   1:  PR[91,1] = PR[90,1] + 32.337;
   1:  PR[91,2] = PR[90,2] + -10.295;
   1:  PR[91,3] = PR[90,3] + 13.551;
   1:L PR[91] R[100]mm/sec CNT100;
   1:  PR[91,1] = PR[90,1] + 32.852;
   1:  PR[91,2] = PR[90,2] + -9.634;
   1:  PR[91,3] = PR[90,3] + 13.557;
   1:L PR[91] R[100]mm/sec CNT100;
   1:  PR[91,1] = PR[90,1] + 33.339;
   1:  PR[91,2] = PR[90,2] + -8.939;
   1:  PR[91,3] = PR[90,3] + 13.562;
   1:L PR[91] R[100]mm/sec CNT100;
   1:  PR[91,1] = PR[90,1] + 33.788;
   1:  PR[91,2] = PR[90,2] + -8.227;
   1:  PR[91,3] = PR[90,3] + 13.568;
   1:L PR[91] R[100]mm/sec CNT100;
   1:  PR[91,1] = PR[90,1] + 34.186;
   1:  PR[91,2] = PR[90,2] + -7.524;
   1:  PR[91,3] = PR[90,3] + 13.574;
   1:L PR[91] R[100]mm/sec CNT100;
   1:  PR[91,1] = PR[90,1] + 34.560;
   1:  PR[91,2] = PR[90,2] + -6.785;
   1:  PR[91,3] = PR[90,3] + 13.579;
   1:L PR[91] R[100]mm/sec CNT100;
   1:  PR[91,1] = PR[90,1] + 34.896;
   1:  PR[91,2] = PR[90,2] + -6.031;
   1:  PR[91,3] = PR[90,3] + 13.584;
   1:L PR[91] R[100]mm/sec CNT100;
   1:  PR[91,1] = PR[90,1] + 35.196;
   1:  PR[91,2] = PR[90,2] + -5.265;
   1:  PR[91,3] = PR[90,3] + 13.590;
   1:L PR[91] R[100]mm/sec CNT100;
   1:  PR[91,1] = PR[90,1] + 35.456;
   1:  PR[91,2] = PR[90,2] + -4.487;
   1:  PR[91,3] = PR[90,3] + 13.595;
   1:L PR[91] R[100]mm/sec CNT100;
   1:  PR[91,1] = PR[90,1] + 35.678;
   1:  PR[91,2] = PR[90,2] + -3.699;
   1:  PR[91,3] = PR[90,3] + 13.600;
   1:L PR[91] R[100]mm/sec CNT100;
   1:  PR[91,1] = PR[90,1] + 35.861;
   1:  PR[91,2] = PR[90,2] + -2.900;
   1:  PR[91,3] = PR[90,3] + 13.606;
   1:L PR[91] R[100]mm/sec CNT100;
   1:  PR[91,1] = PR[90,1] + 36.003;
   1:  PR[91,2] = PR[90,2] + -2.088;
   1:  PR[91,3] = PR[90,3] + 13.611;
   1:L PR[91] R[100]mm/sec CNT100;
   1:  PR[91,1] = PR[90,1] + 36.105;
   1:  PR[91,2] = PR[90,2] + -1.263;
   1:  PR[91,3] = PR[90,3] + 13.617;
   1:L PR[91] R[100]mm/sec CNT100;
   1:  PR[91,1] = PR[90,1] + 36.167;
   1:  PR[91,2] = PR[90,2] + -0.424;
   1:  PR[91,3] = PR[90,3] + 13.622;
   1:L PR[91] R[100]mm/sec CNT100;
   1:  PR[91,1] = PR[90,1] + 36.190;
   1:  PR[91,2] = PR[90,2] + 0.428;
   1:  PR[91,3] = PR[90,3] + 13.628;
   1:L PR[91] R[100]mm/sec CNT100;
   1:  PR[91,1] = PR[90,1] + 36.167;
   1:  PR[91,2] = PR[90,2] + 1.279;
   1:  PR[91,3] = PR[90,3] + 13.633;
   1:L PR[91] R[100]mm/sec CNT100;
   1:  PR[91,1] = PR[90,1] + 36.105;
   1:  PR[91,2] = PR[90,2] + 2.119;
   1:  PR[91,3] = PR[90,3] + 13.639;
   1:L PR[91] R[100]mm/sec CNT100;
   1:  PR[91,1] = PR[90,1] + 36.003;
   1:  PR[91,2] = PR[90,2] + 2.943;
   1:  PR[91,3] = PR[90,3] + 13.644;
   1:L PR[91] R[100]mm/sec CNT100;
   1:  PR[91,1] = PR[90,1] + 35.861;
   1:  PR[91,2] = PR[90,2] + 3.755;
   1:  PR[91,3] = PR[90,3] + 13.650;
   1:L PR[91] R[100]mm/sec CNT100;
   1:  PR[91,1] = PR[90,1] + 35.678;
   1:  PR[91,2] = PR[90,2] + 4.554;
   1:  PR[91,3] = PR[90,3] + 13.655;
   1:L PR[91] R[100]mm/sec CNT100;
   1:  PR[91,1] = PR[90,1] + 35.456;
   1:  PR[91,2] = PR[90,2] + 5.343;
   1:  PR[91,3] = PR[90,3] + 13.660;
   1:L PR[91] R[100]mm/sec CNT100;
   1:  PR[91,1] = PR[90,1] + 35.196;
   1:  PR[91,2] = PR[90,2] + 6.120;
   1:  PR[91,3] = PR[90,3] + 13.666;
   1:L PR[91] R[100]mm/sec CNT100;
   1:  PR[91,1] = PR[90,1] + 34.896;
   1:  PR[91,2] = PR[90,2] + 6.886;
   1:  PR[91,3] = PR[90,3] + 13.671;
   1:L PR[91] R[100]mm/sec CNT100;
   1:  PR[91,1] = PR[90,1] + 34.559;
   1:  PR[91,2] = PR[90,2] + 7.640;
   1:  PR[91,3] = PR[90,3] + 13.677;
   1:L PR[91] R[100]mm/sec CNT100;
   1:  PR[91,1] = PR[90,1] + 34.186;
   1:  PR[91,2] = PR[90,2] + 8.379;
   1:  PR[91,3] = PR[90,3] + 13.682;
   1:L PR[91] R[100]mm/sec CNT100;
   1:  PR[91,1] = PR[90,1] + 33.778;
   1:  PR[91,2] = PR[90,2] + 9.100;
   1:  PR[91,3] = PR[90,3] + 13.687;
   1:L PR[91] R[100]mm/sec CNT100;
   1:  PR[91,1] = PR[90,1] + 33.333;
   1:  PR[91,2] = PR[90,2] + 9.803;
   1:  PR[91,3] = PR[90,3] + 13.693;
   1:L PR[91] R[100]mm/sec CNT100;
   1:  PR[91,1] = PR[90,1] + 32.852;
   1:  PR[91,2] = PR[90,2] + 10.489;
   1:  PR[91,3] = PR[90,3] + 13.698;
   1:L PR[91] R[100]mm/sec CNT100;
   1:  PR[91,1] = PR[90,1] + 32.337;
   1:  PR[91,2] = PR[90,2] + 11.150;
   1:  PR[91,3] = PR[90,3] + 13.704;
   1:L PR[91] R[100]mm/sec CNT100;
   1:  PR[91,1] = PR[90,1] + 31.789;
   1:  PR[91,2] = PR[90,2] + 11.786;
   1:  PR[91,3] = PR[90,3] + 13.709;
   1:L PR[91] R[100]mm/sec CNT100;
   1:  PR[91,1] = PR[90,1] + 31.210;
   1:  PR[91,2] = PR[90,2] + 12.395;
   1:  PR[91,3] = PR[90,3] + 13.715;
   1:L PR[91] R[100]mm/sec CNT100;
   1:  PR[91,1] = PR[90,1] + 30.601;
   1:  PR[91,2] = PR[90,2] + 12.975;
   1:  PR[91,3] = PR[90,3] + 13.720;
   1:L PR[91] R[100]mm/sec CNT100;
   1:  PR[91,1] = PR[90,1] + 29.964;
   1:  PR[91,2] = PR[90,2] + 13.525;
   1:  PR[91,3] = PR[90,3] + 13.726;
   1:L PR[91] R[100]mm/sec CNT100;
   1:  PR[91,1] = PR[90,1] + 29.298;
   1:  PR[91,2] = PR[90,2] + 14.044;
   1:  PR[91,3] = PR[90,3] + 13.731;
   1:L PR[91] R[100]mm/sec CNT100;
   1:  PR[91,1] = PR[90,1] + 28.607;
   1:  PR[91,2] = PR[90,2] + 14.531;
   1:  PR[91,3] = PR[90,3] + 13.737;
   1:L PR[91] R[100]mm/sec CNT100;
   1:  PR[91,1] = PR[90,1] + 27.892;
   1:  PR[91,2] = PR[90,2] + 14.985;
   1:  PR[91,3] = PR[90,3] + 13.742;
   1:L PR[91] R[100]mm/sec CNT100;
   1:  PR[91,1] = PR[90,1] + 27.152;
   1:  PR[91,2] = PR[90,2] + 15.405;
   1:  PR[91,3] = PR[90,3] + 13.748;
   1:L PR[91] R[100]mm/sec CNT100;
   1:  PR[91,1] = PR[90,1] + 26.864;
   1:  PR[91,2] = PR[90,2] + 15.553;
   1:  PR[91,3] = PR[90,3] + 13.753;
   1:L PR[91] R[100]mm/sec CNT100;
   1:  PR[91,1] = PR[90,1] + 26.394;
   1:  PR[91,2] = PR[90,2] + 15.789;
   1:  PR[91,3] = PR[90,3] + 13.756;
   1:L PR[91] R[100]mm/sec CNT100;
   1:  PR[91,1] = PR[90,1] + 25.614;
   1:  PR[91,2] = PR[90,2] + 16.137;
   1:  PR[91,3] = PR[90,3] + 13.759;
   1:L PR[91] R[100]mm/sec CNT100;
   1:  PR[91,1] = PR[90,1] + 24.816;
   1:  PR[91,2] = PR[90,2] + 16.448;
   1:  PR[91,3] = PR[90,3] + 13.765;
   1:L PR[91] R[100]mm/sec CNT100;
   1:  PR[91,1] = PR[90,1] + 24.003;
   1:  PR[91,2] = PR[90,2] + 16.721;
   1:  PR[91,3] = PR[90,3] + 13.770;
   1:L PR[91] R[100]mm/sec CNT100;
   1:  PR[91,1] = PR[90,1] + 23.176;
   1:  PR[91,2] = PR[90,2] + 16.954;
   1:  PR[91,3] = PR[90,3] + 13.776;
   1:L PR[91] R[100]mm/sec CNT100;
   1:  PR[91,1] = PR[90,1] + 22.334;
   1:  PR[91,2] = PR[90,2] + 17.149;
   1:  PR[91,3] = PR[90,3] + 13.781;
   1:L PR[91] R[100]mm/sec CNT100;
   1:  PR[91,1] = PR[90,1] + 21.481;
   1:  PR[91,2] = PR[90,2] + 17.302;
   1:  PR[91,3] = PR[90,3] + 13.787;
   1:L PR[91] R[100]mm/sec CNT100;
   1:  PR[91,1] = PR[90,1] + 20.619;
   1:  PR[91,2] = PR[90,2] + 17.414;
   1:  PR[91,3] = PR[90,3] + 13.793;
   1:L PR[91] R[100]mm/sec CNT100;
   1:  PR[91,1] = PR[90,1] + 20.067;
   1:  PR[91,2] = PR[90,2] + 17.460;
   1:  PR[91,3] = PR[90,3] + 13.799;
   1:L PR[91] R[100]mm/sec CNT100;
   1:  PR[91,1] = PR[90,1] + 19.753;
   1:  PR[91,2] = PR[90,2] + 17.485;
   1:  PR[91,3] = PR[90,3] + 13.802;
   1:L PR[91] R[100]mm/sec CNT100;
   1:  PR[91,1] = PR[90,1] + 18.879;
   1:  PR[91,2] = PR[90,2] + 17.513;
   1:  PR[91,3] = PR[90,3] + 13.804;
   1:L PR[91] R[100]mm/sec CNT100;
   1:  PR[91,1] = PR[90,1] + 18.005;
   1:  PR[91,2] = PR[90,2] + 17.499;
   1:  PR[91,3] = PR[90,3] + 13.810;
   1:L PR[91] R[100]mm/sec CNT100;
   1:  PR[91,1] = PR[90,1] + 17.130;
   1:  PR[91,2] = PR[90,2] + 17.442;
   1:  PR[91,3] = PR[90,3] + 13.816;
   1:L PR[91] R[100]mm/sec CNT100;
   1:  PR[91,1] = PR[90,1] + 16.258;
   1:  PR[91,2] = PR[90,2] + 17.343;
   1:  PR[91,3] = PR[90,3] + 13.821;
   1:L PR[91] R[100]mm/sec CNT100;
   1:  PR[91,1] = PR[90,1] + 15.371;
   1:  PR[91,2] = PR[90,2] + 17.197;
   1:  PR[91,3] = PR[90,3] + 13.827;
   1:L PR[91] R[100]mm/sec CNT100;
   1:  PR[91,1] = PR[90,1] + 14.525;
   1:  PR[91,2] = PR[90,2] + 17.016;
   1:  PR[91,3] = PR[90,3] + 13.833;
   1:L PR[91] R[100]mm/sec CNT100;
   1:  PR[91,1] = PR[90,1] + 13.668;
   1:  PR[91,2] = PR[90,2] + 16.789;
   1:  PR[91,3] = PR[90,3] + 13.839;
   1:L PR[91] R[100]mm/sec CNT100;
   1:  PR[91,1] = PR[90,1] + 12.821;
   1:  PR[91,2] = PR[90,2] + 16.520;
   1:  PR[91,3] = PR[90,3] + 13.845;
   1:L PR[91] R[100]mm/sec CNT100;
   1:  PR[91,1] = PR[90,1] + 11.988;
   1:  PR[91,2] = PR[90,2] + 16.209;
   1:  PR[91,3] = PR[90,3] + 13.850;
   1:L PR[91] R[100]mm/sec CNT100;
   1:  PR[91,1] = PR[90,1] + 11.168;
   1:  PR[91,2] = PR[90,2] + 15.858;
   1:  PR[91,3] = PR[90,3] + 13.856;
   1:L PR[91] R[100]mm/sec CNT100;
   1:  PR[91,1] = PR[90,1] + 10.890;
   1:  PR[91,2] = PR[90,2] + 15.724;
   1:  PR[91,3] = PR[90,3] + 13.862;
   1:L PR[91] R[100]mm/sec CNT100;
   1:  PR[91,1] = PR[90,1] + 10.371;
   1:  PR[91,2] = PR[90,2] + 15.468;
   1:  PR[91,3] = PR[90,3] + 13.864;
   1:L PR[91] R[100]mm/sec CNT100;
   1:  PR[91,1] = PR[90,1] + 9.590;
   1:  PR[91,2] = PR[90,2] + 15.037;
   1:  PR[91,3] = PR[90,3] + 13.868;
   1:L PR[91] R[100]mm/sec CNT100;
   1:  PR[91,1] = PR[90,1] + 8.823;
   1:  PR[91,2] = PR[90,2] + 14.562;
   1:  PR[91,3] = PR[90,3] + 13.874;
   1:L PR[91] R[100]mm/sec CNT100;
   1:  PR[91,1] = PR[90,1] + 8.157;
   1:  PR[91,2] = PR[90,2] + 14.105;
   1:  PR[91,3] = PR[90,3] + 13.880;
   1:L PR[91] R[100]mm/sec CNT100;
   1:  PR[91,1] = PR[90,1] + 7.356;
   1:  PR[91,2] = PR[90,2] + 13.495;
   1:  PR[91,3] = PR[90,3] + 13.885;
   1:L PR[91] R[100]mm/sec CNT100;
   1:  PR[91,1] = PR[90,1] + 6.666;
   1:  PR[91,2] = PR[90,2] + 12.906;
   1:  PR[91,3] = PR[90,3] + 13.892;
   1:L PR[91] R[100]mm/sec CNT100;
   1:  PR[91,1] = PR[90,1] + 6.298;
   1:  PR[91,2] = PR[90,2] + 12.563;
   1:  PR[91,3] = PR[90,3] + 13.897;
   1:L PR[91] R[100]mm/sec CNT100;
   1:  PR[91,1] = PR[90,1] + 5.727;
   1:  PR[91,2] = PR[90,2] + 11.992;
   1:  PR[91,3] = PR[90,3] + 13.901;
   1:L PR[91] R[100]mm/sec CNT100;
   1:  PR[91,1] = PR[90,1] + 5.186;
   1:  PR[91,2] = PR[90,2] + 11.396;
   1:  PR[91,3] = PR[90,3] + 13.906;
   1:L PR[91] R[100]mm/sec CNT100;
   1:  PR[91,1] = PR[90,1] + 4.817;
   1:  PR[91,2] = PR[90,2] + 10.959;
   1:  PR[91,3] = PR[90,3] + 13.911;
   1:L PR[91] R[100]mm/sec CNT100;
   1:  PR[91,1] = PR[90,1] + 4.192;
   1:  PR[91,2] = PR[90,2] + 10.135;
   1:  PR[91,3] = PR[90,3] + 13.915;
   1:L PR[91] R[100]mm/sec CNT100;
   1:  PR[91,1] = PR[90,1] + 3.772;
   1:  PR[91,2] = PR[90,2] + 9.523;
   1:  PR[91,3] = PR[90,3] + 13.922;
   1:L PR[91] R[100]mm/sec CNT100;
   1:  PR[91,1] = PR[90,1] + 3.309;
   1:  PR[91,2] = PR[90,2] + 8.774;
   1:  PR[91,3] = PR[90,3] + 13.927;
   1:L PR[91] R[100]mm/sec CNT100;
   1:  PR[91,1] = PR[90,1] + 2.885;
   1:  PR[91,2] = PR[90,2] + 8.008;
   1:  PR[91,3] = PR[90,3] + 13.932;
   1:L PR[91] R[100]mm/sec CNT100;
   1:  PR[91,1] = PR[90,1] + 2.385;
   1:  PR[91,2] = PR[90,2] + 7.023;
   1:  PR[91,3] = PR[90,3] + 13.938;
   1:L PR[91] R[100]mm/sec CNT100;
   1:  PR[91,1] = PR[90,1] + 2.105;
   1:  PR[91,2] = PR[90,2] + 6.621;
   1:  PR[91,3] = PR[90,3] + 13.945;
   1:L PR[91] R[100]mm/sec CNT100;
   1:  PR[91,1] = PR[90,1] + 1.841;
   1:  PR[91,2] = PR[90,2] + 6.326;
   1:  PR[91,3] = PR[90,3] + 13.949;
   1:L PR[91] R[100]mm/sec CNT100;
   1:  PR[91,1] = PR[90,1] + 1.518;
   1:  PR[91,2] = PR[90,2] + 6.046;
   1:  PR[91,3] = PR[90,3] + 13.951;
   1:L PR[91] R[100]mm/sec CNT100;
   1:  PR[91,1] = PR[90,1] + 1.046;
   1:  PR[91,2] = PR[90,2] + 5.756;
   1:  PR[91,3] = PR[90,3] + 13.954;
   1:L PR[91] R[100]mm/sec CNT100;
   1:  PR[91,1] = PR[90,1] + 0.789;
   1:  PR[91,2] = PR[90,2] + 5.645;
   1:  PR[91,3] = PR[90,3] + 13.958;
   1:L PR[91] R[100]mm/sec CNT100;
   1:  PR[91,1] = PR[90,1] + 0.396;
   1:  PR[91,2] = PR[90,2] + 5.532;
   1:  PR[91,3] = PR[90,3] + 13.960;
   1:L PR[91] R[100]mm/sec CNT100;
   1:  PR[91,1] = PR[90,1] + -0.008;
   1:  PR[91,2] = PR[90,2] + 5.483;
   1:  PR[91,3] = PR[90,3] + 13.962;
   1:L PR[91] R[100]mm/sec CNT100;
   1:  PR[91,1] = PR[90,1] + -0.238;
   1:  PR[91,2] = PR[90,2] + 5.484;
   1:  PR[91,3] = PR[90,3] + 13.965;
   1:L PR[91] R[100]mm/sec CNT100;
   1:  PR[91,1] = PR[90,1] + -0.633;
   1:  PR[91,2] = PR[90,2] + 5.532;
   1:  PR[91,3] = PR[90,3] + 13.966;
   1:L PR[91] R[100]mm/sec CNT100;
   1:  PR[91,1] = PR[90,1] + -0.865;
   1:  PR[91,2] = PR[90,2] + 5.591;
   1:  PR[91,3] = PR[90,3] + 13.969;
   1:L PR[91] R[100]mm/sec CNT100;
   1:  PR[91,1] = PR[90,1] + -1.055;
   1:  PR[91,2] = PR[90,2] + 5.655;
   1:  PR[91,3] = PR[90,3] + 13.971;
   1:L PR[91] R[100]mm/sec CNT100;
   1:  PR[91,1] = PR[90,1] + -1.421;
   1:  PR[91,2] = PR[90,2] + 5.826;
   1:  PR[91,3] = PR[90,3] + 13.972;
   1:L PR[91] R[100]mm/sec CNT100;
   1:  PR[91,1] = PR[90,1] + -1.767;
   1:  PR[91,2] = PR[90,2] + 6.053;
   1:  PR[91,3] = PR[90,3] + 13.975;
   1:L PR[91] R[100]mm/sec CNT100;
   1:  PR[91,1] = PR[90,1] + -2.029;
   1:  PR[91,2] = PR[90,2] + 6.277;
   1:  PR[91,3] = PR[90,3] + 13.977;
   1:L PR[91] R[100]mm/sec CNT100;
   1:  PR[91,1] = PR[90,1] + -2.346;
   1:  PR[91,2] = PR[90,2] + 6.622;
   1:  PR[91,3] = PR[90,3] + 13.979;
   1:L PR[91] R[100]mm/sec CNT100;
   1:  PR[91,1] = PR[90,1] + -2.615;
   1:  PR[91,2] = PR[90,2] + 7.005;
   1:  PR[91,3] = PR[90,3] + 13.983;
   1:L PR[91] R[100]mm/sec CNT100;
   1:  PR[91,1] = PR[90,1] + -3.128;
   1:  PR[91,2] = PR[90,2] + 8.018;
   1:  PR[91,3] = PR[90,3] + 13.986;
   1:L PR[91] R[100]mm/sec CNT100;
   1:  PR[91,1] = PR[90,1] + -3.562;
   1:  PR[91,2] = PR[90,2] + 8.804;
   1:  PR[91,3] = PR[90,3] + 13.993;
   1:L PR[91] R[100]mm/sec CNT100;
   1:  PR[91,1] = PR[90,1] + -4.015;
   1:  PR[91,2] = PR[90,2] + 9.537;
   1:  PR[91,3] = PR[90,3] + 13.999;
   1:L PR[91] R[100]mm/sec CNT100;
   1:  PR[91,1] = PR[90,1] + -4.434;
   1:  PR[91,2] = PR[90,2] + 10.149;
   1:  PR[91,3] = PR[90,3] + 14.005;
   1:L PR[91] R[100]mm/sec CNT100;
   1:  PR[91,1] = PR[90,1] + -5.061;
   1:  PR[91,2] = PR[90,2] + 10.971;
   1:  PR[91,3] = PR[90,3] + 14.009;
   1:L PR[91] R[100]mm/sec CNT100;
   1:  PR[91,1] = PR[90,1] + -5.426;
   1:  PR[91,2] = PR[90,2] + 11.402;
   1:  PR[91,3] = PR[90,3] + 14.016;
   1:L PR[91] R[100]mm/sec CNT100;
   1:  PR[91,1] = PR[90,1] + -6.258;
   1:  PR[91,2] = PR[90,2] + 12.293;
   1:  PR[91,3] = PR[90,3] + 14.020;
   1:L PR[91] R[100]mm/sec CNT100;
   1:  PR[91,1] = PR[90,1] + -7.138;
   1:  PR[91,2] = PR[90,2] + 13.109;
   1:  PR[91,3] = PR[90,3] + 14.028;
   1:L PR[91] R[100]mm/sec CNT100;
   1:  PR[91,1] = PR[90,1] + -7.601;
   1:  PR[91,2] = PR[90,2] + 13.498;
   1:  PR[91,3] = PR[90,3] + 14.036;
   1:L PR[91] R[100]mm/sec CNT100;
   1:  PR[91,1] = PR[90,1] + -8.326;
   1:  PR[91,2] = PR[90,2] + 14.053;
   1:  PR[91,3] = PR[90,3] + 14.040;
   1:L PR[91] R[100]mm/sec CNT100;
   1:  PR[91,1] = PR[90,1] + -9.078;
   1:  PR[91,2] = PR[90,2] + 14.571;
   1:  PR[91,3] = PR[90,3] + 14.046;
   1:L PR[91] R[100]mm/sec CNT100;
   1:  PR[91,1] = PR[90,1] + -9.837;
   1:  PR[91,2] = PR[90,2] + 15.040;
   1:  PR[91,3] = PR[90,3] + 14.052;
   1:L PR[91] R[100]mm/sec CNT100;
   1:  PR[91,1] = PR[90,1] + -10.425;
   1:  PR[91,2] = PR[90,2] + 15.367;
   1:  PR[91,3] = PR[90,3] + 14.058;
   1:L PR[91] R[100]mm/sec CNT100;
   1:  PR[91,1] = PR[90,1] + -11.419;
   1:  PR[91,2] = PR[90,2] + 15.863;
   1:  PR[91,3] = PR[90,3] + 14.062;
   1:L PR[91] R[100]mm/sec CNT100;
   1:  PR[91,1] = PR[90,1] + -12.234;
   1:  PR[91,2] = PR[90,2] + 16.213;
   1:  PR[91,3] = PR[90,3] + 14.069;
   1:L PR[91] R[100]mm/sec CNT100;
   1:  PR[91,1] = PR[90,1] + -13.065;
   1:  PR[91,2] = PR[90,2] + 16.523;
   1:  PR[91,3] = PR[90,3] + 14.075;
   1:L PR[91] R[100]mm/sec CNT100;
   1:  PR[91,1] = PR[90,1] + -14.084;
   1:  PR[91,2] = PR[90,2] + 16.839;
   1:  PR[91,3] = PR[90,3] + 14.081;
   1:L PR[91] R[100]mm/sec CNT100;
   1:  PR[91,1] = PR[90,1] + -14.770;
   1:  PR[91,2] = PR[90,2] + 17.018;
   1:  PR[91,3] = PR[90,3] + 14.088;
   1:L PR[91] R[100]mm/sec CNT100;
   1:  PR[91,1] = PR[90,1] + -15.636;
   1:  PR[91,2] = PR[90,2] + 17.202;
   1:  PR[91,3] = PR[90,3] + 14.092;
   1:L PR[91] R[100]mm/sec CNT100;
   1:  PR[91,1] = PR[90,1] + -16.504;
   1:  PR[91,2] = PR[90,2] + 17.344;
   1:  PR[91,3] = PR[90,3] + 14.098;
   1:L PR[91] R[100]mm/sec CNT100;
   1:  PR[91,1] = PR[90,1] + -17.376;
   1:  PR[91,2] = PR[90,2] + 17.443;
   1:  PR[91,3] = PR[90,3] + 14.104;
   1:L PR[91] R[100]mm/sec CNT100;
   1:  PR[91,1] = PR[90,1] + -18.251;
   1:  PR[91,2] = PR[90,2] + 17.499;
   1:  PR[91,3] = PR[90,3] + 14.110;
   1:L PR[91] R[100]mm/sec CNT100;
   1:  PR[91,1] = PR[90,1] + -18.743;
   1:  PR[91,2] = PR[90,2] + 17.508;
   1:  PR[91,3] = PR[90,3] + 14.116;
   1:L PR[91] R[100]mm/sec CNT100;
   1:  PR[91,1] = PR[90,1] + -19.123;
   1:  PR[91,2] = PR[90,2] + 17.513;
   1:  PR[91,3] = PR[90,3] + 14.119;
   1:L PR[91] R[100]mm/sec CNT100;
   1:  PR[91,1] = PR[90,1] + -19.996;
   1:  PR[91,2] = PR[90,2] + 17.484;
   1:  PR[91,3] = PR[90,3] + 14.121;
   1:L PR[91] R[100]mm/sec CNT100;
   1:  PR[91,1] = PR[90,1] + -20.863;
   1:  PR[91,2] = PR[90,2] + 17.413;
   1:  PR[91,3] = PR[90,3] + 14.127;
   1:L PR[91] R[100]mm/sec CNT100;
   1:  PR[91,1] = PR[90,1] + -21.725;
   1:  PR[91,2] = PR[90,2] + 17.301;
   1:  PR[91,3] = PR[90,3] + 14.133;
   1:L PR[91] R[100]mm/sec CNT100;
   1:  PR[91,1] = PR[90,1] + -22.577;
   1:  PR[91,2] = PR[90,2] + 17.148;
   1:  PR[91,3] = PR[90,3] + 14.138;
   1:L PR[91] R[100]mm/sec CNT100;
   1:  PR[91,1] = PR[90,1] + -23.424;
   1:  PR[91,2] = PR[90,2] + 16.953;
   1:  PR[91,3] = PR[90,3] + 14.144;
   1:L PR[91] R[100]mm/sec CNT100;
   1:  PR[91,1] = PR[90,1] + -24.247;
   1:  PR[91,2] = PR[90,2] + 16.720;
   1:  PR[91,3] = PR[90,3] + 14.150;
   1:L PR[91] R[100]mm/sec CNT100;
   1:  PR[91,1] = PR[90,1] + -25.059;
   1:  PR[91,2] = PR[90,2] + 16.448;
   1:  PR[91,3] = PR[90,3] + 14.155;
   1:L PR[91] R[100]mm/sec CNT100;
   1:  PR[91,1] = PR[90,1] + -25.856;
   1:  PR[91,2] = PR[90,2] + 16.137;
   1:  PR[91,3] = PR[90,3] + 14.161;
   1:L PR[91] R[100]mm/sec CNT100;
   1:  PR[91,1] = PR[90,1] + -26.635;
   1:  PR[91,2] = PR[90,2] + 15.788;
   1:  PR[91,3] = PR[90,3] + 14.167;
   1:L PR[91] R[100]mm/sec CNT100;
   1:  PR[91,1] = PR[90,1] + -27.104;
   1:  PR[91,2] = PR[90,2] + 15.551;
   1:  PR[91,3] = PR[90,3] + 14.172;
   1:L PR[91] R[100]mm/sec CNT100;
   1:  PR[91,1] = PR[90,1] + -27.393;
   1:  PR[91,2] = PR[90,2] + 15.403;
   1:  PR[91,3] = PR[90,3] + 14.176;
   1:L PR[91] R[100]mm/sec CNT100;
   1:  PR[91,1] = PR[90,1] + -28.133;
   1:  PR[91,2] = PR[90,2] + 14.983;
   1:  PR[91,3] = PR[90,3] + 14.178;
   1:L PR[91] R[100]mm/sec CNT100;
   1:  PR[91,1] = PR[90,1] + -28.848;
   1:  PR[91,2] = PR[90,2] + 14.528;
   1:  PR[91,3] = PR[90,3] + 14.183;
   1:L PR[91] R[100]mm/sec CNT100;
   1:  PR[91,1] = PR[90,1] + -29.539;
   1:  PR[91,2] = PR[90,2] + 14.041;
   1:  PR[91,3] = PR[90,3] + 14.189;
   1:L PR[91] R[100]mm/sec CNT100;
   1:  PR[91,1] = PR[90,1] + -30.204;
   1:  PR[91,2] = PR[90,2] + 13.522;
   1:  PR[91,3] = PR[90,3] + 14.194;
   1:L PR[91] R[100]mm/sec CNT100;
   1:  PR[91,1] = PR[90,1] + -30.842;
   1:  PR[91,2] = PR[90,2] + 12.972;
   1:  PR[91,3] = PR[90,3] + 14.200;
   1:L PR[91] R[100]mm/sec CNT100;
   1:  PR[91,1] = PR[90,1] + -31.451;
   1:  PR[91,2] = PR[90,2] + 12.393;
   1:  PR[91,3] = PR[90,3] + 14.205;
   1:L PR[91] R[100]mm/sec CNT100;
   1:  PR[91,1] = PR[90,1] + -32.029;
   1:  PR[91,2] = PR[90,2] + 11.785;
   1:  PR[91,3] = PR[90,3] + 14.211;
   1:L PR[91] R[100]mm/sec CNT100;
   1:  PR[91,1] = PR[90,1] + -32.577;
   1:  PR[91,2] = PR[90,2] + 11.151;
   1:  PR[91,3] = PR[90,3] + 14.216;
   1:L PR[91] R[100]mm/sec CNT100;
   1:  PR[91,1] = PR[90,1] + -33.092;
   1:  PR[91,2] = PR[90,2] + 10.491;
   1:  PR[91,3] = PR[90,3] + 14.222;
   1:L PR[91] R[100]mm/sec CNT100;
   1:  PR[91,1] = PR[90,1] + -33.579;
   1:  PR[91,2] = PR[90,2] + 9.797;
   1:  PR[91,3] = PR[90,3] + 14.227;
   1:L PR[91] R[100]mm/sec CNT100;
   1:  PR[91,1] = PR[90,1] + -34.027;
   1:  PR[91,2] = PR[90,2] + 9.084;
   1:  PR[91,3] = PR[90,3] + 14.233;
   1:L PR[91] R[100]mm/sec CNT100;
   1:  PR[91,1] = PR[90,1] + -34.425;
   1:  PR[91,2] = PR[90,2] + 8.381;
   1:  PR[91,3] = PR[90,3] + 14.239;
   1:L PR[91] R[100]mm/sec CNT100;
   1:  PR[91,1] = PR[90,1] + -34.798;
   1:  PR[91,2] = PR[90,2] + 7.639;
   1:  PR[91,3] = PR[90,3] + 14.244;
   1:L PR[91] R[100]mm/sec CNT100;
   1:  PR[91,1] = PR[90,1] + -35.135;
   1:  PR[91,2] = PR[90,2] + 6.883;
   1:  PR[91,3] = PR[90,3] + 14.249;
   1:L PR[91] R[100]mm/sec CNT100;
   1:  PR[91,1] = PR[90,1] + -35.434;
   1:  PR[91,2] = PR[90,2] + 6.114;
   1:  PR[91,3] = PR[90,3] + 14.255;
   1:L PR[91] R[100]mm/sec CNT100;
   1:  PR[91,1] = PR[90,1] + -35.695;
   1:  PR[91,2] = PR[90,2] + 5.335;
   1:  PR[91,3] = PR[90,3] + 14.260;
   1:L PR[91] R[100]mm/sec CNT100;
   1:  PR[91,1] = PR[90,1] + -35.917;
   1:  PR[91,2] = PR[90,2] + 4.546;
   1:  PR[91,3] = PR[90,3] + 14.265;
   1:L PR[91] R[100]mm/sec CNT100;
   1:  PR[91,1] = PR[90,1] + -36.099;
   1:  PR[91,2] = PR[90,2] + 3.748;
   1:  PR[91,3] = PR[90,3] + 14.271;
   1:L PR[91] R[100]mm/sec CNT100;
   1:  PR[91,1] = PR[90,1] + -36.242;
   1:  PR[91,2] = PR[90,2] + 2.938;
   1:  PR[91,3] = PR[90,3] + 14.276;
   1:L PR[91] R[100]mm/sec CNT100;
   1:  PR[91,1] = PR[90,1] + -36.344;
   1:  PR[91,2] = PR[90,2] + 2.116;
   1:  PR[91,3] = PR[90,3] + 14.282;
   1:L PR[91] R[100]mm/sec CNT100;
   1:  PR[91,1] = PR[90,1] + -36.405;
   1:  PR[91,2] = PR[90,2] + 1.278;
   1:  PR[91,3] = PR[90,3] + 14.287;
   1:L PR[91] R[100]mm/sec CNT100;
   1:  PR[91,1] = PR[90,1] + -36.428;
   1:  PR[91,2] = PR[90,2] + 0.428;
   1:  PR[91,3] = PR[90,3] + 14.293;
   1:L PR[91] R[100]mm/sec CNT100;
   1:  PR[91,1] = PR[90,1] + -36.405;
   1:  PR[91,2] = PR[90,2] + -0.423;
   1:  PR[91,3] = PR[90,3] + 14.298;
   1:L PR[91] R[100]mm/sec CNT100;
   1:  PR[91,1] = PR[90,1] + -36.344;
   1:  PR[91,2] = PR[90,2] + -1.261;
   1:  PR[91,3] = PR[90,3] + 14.304;
   1:L PR[91] R[100]mm/sec CNT100;
   1:  PR[91,1] = PR[90,1] + -36.242;
   1:  PR[91,2] = PR[90,2] + -2.083;
   1:  PR[91,3] = PR[90,3] + 14.309;
   1:L PR[91] R[100]mm/sec CNT100;
   1:  PR[91,1] = PR[90,1] + -36.099;
   1:  PR[91,2] = PR[90,2] + -2.892;
   1:  PR[91,3] = PR[90,3] + 14.315;
   1:L PR[91] R[100]mm/sec CNT100;
   1:  PR[91,1] = PR[90,1] + -35.917;
   1:  PR[91,2] = PR[90,2] + -3.691;
   1:  PR[91,3] = PR[90,3] + 14.320;
   1:L PR[91] R[100]mm/sec CNT100;
   1:  PR[91,1] = PR[90,1] + -35.695;
   1:  PR[91,2] = PR[90,2] + -4.480;
   1:  PR[91,3] = PR[90,3] + 14.325;
   1:L PR[91] R[100]mm/sec CNT100;
   1:  PR[91,1] = PR[90,1] + -35.434;
   1:  PR[91,2] = PR[90,2] + -5.259;
   1:  PR[91,3] = PR[90,3] + 14.331;
   1:L PR[91] R[100]mm/sec CNT100;
   1:  PR[91,1] = PR[90,1] + -35.135;
   1:  PR[91,2] = PR[90,2] + -6.028;
   1:  PR[91,3] = PR[90,3] + 14.336;
   1:L PR[91] R[100]mm/sec CNT100;
   1:  PR[91,1] = PR[90,1] + -34.798;
   1:  PR[91,2] = PR[90,2] + -6.784;
   1:  PR[91,3] = PR[90,3] + 14.342;
   1:L PR[91] R[100]mm/sec CNT100;
   1:  PR[91,1] = PR[90,1] + -34.425;
   1:  PR[91,2] = PR[90,2] + -7.525;
   1:  PR[91,3] = PR[90,3] + 14.347;
   1:L PR[91] R[100]mm/sec CNT100;
   1:  PR[91,1] = PR[90,1] + -34.027;
   1:  PR[91,2] = PR[90,2] + -8.229;
   1:  PR[91,3] = PR[90,3] + 14.352;
   1:L PR[91] R[100]mm/sec CNT100;
   1:  PR[91,1] = PR[90,1] + -33.573;
   1:  PR[91,2] = PR[90,2] + -8.951;
   1:  PR[91,3] = PR[90,3] + 14.358;
   1:L PR[91] R[100]mm/sec CNT100;
   1:  PR[91,1] = PR[90,1] + -33.092;
   1:  PR[91,2] = PR[90,2] + -9.636;
   1:  PR[91,3] = PR[90,3] + 14.363;
   1:L PR[91] R[100]mm/sec CNT100;
   1:  PR[91,1] = PR[90,1] + -32.577;
   1:  PR[91,2] = PR[90,2] + -10.296;
   1:  PR[91,3] = PR[90,3] + 14.369;
   1:L PR[91] R[100]mm/sec CNT100;
   1:  PR[91,1] = PR[90,1] + -32.029;
   1:  PR[91,2] = PR[90,2] + -10.930;
   1:  PR[91,3] = PR[90,3] + 14.374;
   1:L PR[91] R[100]mm/sec CNT100;
   1:  PR[91,1] = PR[90,1] + -31.451;
   1:  PR[91,2] = PR[90,2] + -11.537;
   1:  PR[91,3] = PR[90,3] + 14.380;
   1:L PR[91] R[100]mm/sec CNT100;
   1:  PR[91,1] = PR[90,1] + -30.842;
   1:  PR[91,2] = PR[90,2] + -12.117;
   1:  PR[91,3] = PR[90,3] + 14.385;
   1:L PR[91] R[100]mm/sec CNT100;
   1:  PR[91,1] = PR[90,1] + -30.204;
   1:  PR[91,2] = PR[90,2] + -12.667;
   1:  PR[91,3] = PR[90,3] + 14.391;
   1:L PR[91] R[100]mm/sec CNT100;
   1:  PR[91,1] = PR[90,1] + -29.539;
   1:  PR[91,2] = PR[90,2] + -13.186;
   1:  PR[91,3] = PR[90,3] + 14.396;
   1:L PR[91] R[100]mm/sec CNT100;
   1:  PR[91,1] = PR[90,1] + -28.848;
   1:  PR[91,2] = PR[90,2] + -13.673;
   1:  PR[91,3] = PR[90,3] + 14.402;
   1:L PR[91] R[100]mm/sec CNT100;
   1:  PR[91,1] = PR[90,1] + -28.132;
   1:  PR[91,2] = PR[90,2] + -14.128;
   1:  PR[91,3] = PR[90,3] + 14.407;
   1:L PR[91] R[100]mm/sec CNT100;
   1:  PR[91,1] = PR[90,1] + -27.799;
   1:  PR[91,2] = PR[90,2] + -14.319;
   1:  PR[91,3] = PR[90,3] + 14.413;
   1:L PR[91] R[100]mm/sec CNT100;
   1:  PR[91,1] = PR[90,1] + -27.395;
   1:  PR[91,2] = PR[90,2] + -14.548;
   1:  PR[91,3] = PR[90,3] + 14.415;
   1:L PR[91] R[100]mm/sec CNT100;
   1:  PR[91,1] = PR[90,1] + -26.635;
   1:  PR[91,2] = PR[90,2] + -14.933;
   1:  PR[91,3] = PR[90,3] + 14.418;
   1:L PR[91] R[100]mm/sec CNT100;
   1:  PR[91,1] = PR[90,1] + -25.856;
   1:  PR[91,2] = PR[90,2] + -15.281;
   1:  PR[91,3] = PR[90,3] + 14.424;
   1:L PR[91] R[100]mm/sec CNT100;
   1:  PR[91,1] = PR[90,1] + -25.059;
   1:  PR[91,2] = PR[90,2] + -15.593;
   1:  PR[91,3] = PR[90,3] + 14.430;
   1:L PR[91] R[100]mm/sec CNT100;
   1:  PR[91,1] = PR[90,1] + -24.247;
   1:  PR[91,2] = PR[90,2] + -15.865;
   1:  PR[91,3] = PR[90,3] + 14.435;
   1:L PR[91] R[100]mm/sec CNT100;
   1:  PR[91,1] = PR[90,1] + -23.420;
   1:  PR[91,2] = PR[90,2] + -16.099;
   1:  PR[91,3] = PR[90,3] + 14.441;
   1:L PR[91] R[100]mm/sec CNT100;
   1:  PR[91,1] = PR[90,1] + -22.578;
   1:  PR[91,2] = PR[90,2] + -16.293;
   1:  PR[91,3] = PR[90,3] + 14.446;
   1:L PR[91] R[100]mm/sec CNT100;
   1:  PR[91,1] = PR[90,1] + -21.725;
   1:  PR[91,2] = PR[90,2] + -16.446;
   1:  PR[91,3] = PR[90,3] + 14.452;
   1:L PR[91] R[100]mm/sec CNT100;
   1:  PR[91,1] = PR[90,1] + -20.863;
   1:  PR[91,2] = PR[90,2] + -16.558;
   1:  PR[91,3] = PR[90,3] + 14.458;
   1:L PR[91] R[100]mm/sec CNT100;
   1:  PR[91,1] = PR[90,1] + -19.995;
   1:  PR[91,2] = PR[90,2] + -16.629;
   1:  PR[91,3] = PR[90,3] + 14.463;
   1:L PR[91] R[100]mm/sec CNT100;
   1:  PR[91,1] = PR[90,1] + -19.527;
   1:  PR[91,2] = PR[90,2] + -16.646;
   1:  PR[91,3] = PR[90,3] + 14.469;
   1:L PR[91] R[100]mm/sec CNT100;
   1:  PR[91,1] = PR[90,1] + -19.125;
   1:  PR[91,2] = PR[90,2] + -16.658;
   1:  PR[91,3] = PR[90,3] + 14.472;
   1:L PR[91] R[100]mm/sec CNT100;
   1:  PR[91,1] = PR[90,1] + -18.250;
   1:  PR[91,2] = PR[90,2] + -16.644;
   1:  PR[91,3] = PR[90,3] + 14.475;
   1:L PR[91] R[100]mm/sec CNT100;
   1:  PR[91,1] = PR[90,1] + -17.376;
   1:  PR[91,2] = PR[90,2] + -16.588;
   1:  PR[91,3] = PR[90,3] + 14.481;
   1:L PR[91] R[100]mm/sec CNT100;
   1:  PR[91,1] = PR[90,1] + -16.504;
   1:  PR[91,2] = PR[90,2] + -16.489;
   1:  PR[91,3] = PR[90,3] + 14.486;
   1:L PR[91] R[100]mm/sec CNT100;
   1:  PR[91,1] = PR[90,1] + -15.615;
   1:  PR[91,2] = PR[90,2] + -16.343;
   1:  PR[91,3] = PR[90,3] + 14.492;
   1:L PR[91] R[100]mm/sec CNT100;
   1:  PR[91,1] = PR[90,1] + -14.770;
   1:  PR[91,2] = PR[90,2] + -16.163;
   1:  PR[91,3] = PR[90,3] + 14.498;
   1:L PR[91] R[100]mm/sec CNT100;
   1:  PR[91,1] = PR[90,1] + -13.913;
   1:  PR[91,2] = PR[90,2] + -15.937;
   1:  PR[91,3] = PR[90,3] + 14.504;
   1:L PR[91] R[100]mm/sec CNT100;
   1:  PR[91,1] = PR[90,1] + -13.067;
   1:  PR[91,2] = PR[90,2] + -15.669;
   1:  PR[91,3] = PR[90,3] + 14.510;
   1:L PR[91] R[100]mm/sec CNT100;
   1:  PR[91,1] = PR[90,1] + -12.234;
   1:  PR[91,2] = PR[90,2] + -15.358;
   1:  PR[91,3] = PR[90,3] + 14.515;
   1:L PR[91] R[100]mm/sec CNT100;
   1:  PR[91,1] = PR[90,1] + -11.415;
   1:  PR[91,2] = PR[90,2] + -15.006;
   1:  PR[91,3] = PR[90,3] + 14.521;
   1:L PR[91] R[100]mm/sec CNT100;
   1:  PR[91,1] = PR[90,1] + -11.136;
   1:  PR[91,2] = PR[90,2] + -14.872;
   1:  PR[91,3] = PR[90,3] + 14.527;
   1:L PR[91] R[100]mm/sec CNT100;
   1:  PR[91,1] = PR[90,1] + -10.617;
   1:  PR[91,2] = PR[90,2] + -14.616;
   1:  PR[91,3] = PR[90,3] + 14.529;
   1:L PR[91] R[100]mm/sec CNT100;
   1:  PR[91,1] = PR[90,1] + -9.837;
   1:  PR[91,2] = PR[90,2] + -14.185;
   1:  PR[91,3] = PR[90,3] + 14.533;
   1:L PR[91] R[100]mm/sec CNT100;
   1:  PR[91,1] = PR[90,1] + -9.068;
   1:  PR[91,2] = PR[90,2] + -13.709;
   1:  PR[91,3] = PR[90,3] + 14.539;
   1:L PR[91] R[100]mm/sec CNT100;
   1:  PR[91,1] = PR[90,1] + -8.325;
   1:  PR[91,2] = PR[90,2] + -13.198;
   1:  PR[91,3] = PR[90,3] + 14.545;
   1:L PR[91] R[100]mm/sec CNT100;
   1:  PR[91,1] = PR[90,1] + -7.601;
   1:  PR[91,2] = PR[90,2] + -12.642;
   1:  PR[91,3] = PR[90,3] + 14.550;
   1:L PR[91] R[100]mm/sec CNT100;
   1:  PR[91,1] = PR[90,1] + -7.138;
   1:  PR[91,2] = PR[90,2] + -12.254;
   1:  PR[91,3] = PR[90,3] + 14.556;
   1:L PR[91] R[100]mm/sec CNT100;
   1:  PR[91,1] = PR[90,1] + -6.258;
   1:  PR[91,2] = PR[90,2] + -11.438;
   1:  PR[91,3] = PR[90,3] + 14.560;
   1:L PR[91] R[100]mm/sec CNT100;
   1:  PR[91,1] = PR[90,1] + -5.426;
   1:  PR[91,2] = PR[90,2] + -10.547;
   1:  PR[91,3] = PR[90,3] + 14.568;
   1:L PR[91] R[100]mm/sec CNT100;
   1:  PR[91,1] = PR[90,1] + -5.059;
   1:  PR[91,2] = PR[90,2] + -10.115;
   1:  PR[91,3] = PR[90,3] + 14.576;
   1:L PR[91] R[100]mm/sec CNT100;
   1:  PR[91,1] = PR[90,1] + -4.517;
   1:  PR[91,2] = PR[90,2] + -9.410;
   1:  PR[91,3] = PR[90,3] + 14.580;
   1:L PR[91] R[100]mm/sec CNT100;
   1:  PR[91,1] = PR[90,1] + -4.014;
   1:  PR[91,2] = PR[90,2] + -8.682;
   1:  PR[91,3] = PR[90,3] + 14.586;
   1:L PR[91] R[100]mm/sec CNT100;
   1:  PR[91,1] = PR[90,1] + -3.552;
   1:  PR[91,2] = PR[90,2] + -7.933;
   1:  PR[91,3] = PR[90,3] + 14.592;
   1:L PR[91] R[100]mm/sec CNT100;
   1:  PR[91,1] = PR[90,1] + -3.128;
   1:  PR[91,2] = PR[90,2] + -7.162;
   1:  PR[91,3] = PR[90,3] + 14.597;
   1:L PR[91] R[100]mm/sec CNT100;
   1:  PR[91,1] = PR[90,1] + -2.615;
   1:  PR[91,2] = PR[90,2] + -6.150;
   1:  PR[91,3] = PR[90,3] + 14.603;
   1:L PR[91] R[100]mm/sec CNT100;
   1:  PR[91,1] = PR[90,1] + -2.367;
   1:  PR[91,2] = PR[90,2] + -5.793;
   1:  PR[91,3] = PR[90,3] + 14.611;
   1:L PR[91] R[100]mm/sec CNT100;
   1:  PR[91,1] = PR[90,1] + -2.081;
   1:  PR[91,2] = PR[90,2] + -5.471;
   1:  PR[91,3] = PR[90,3] + 14.613;
   1:L PR[91] R[100]mm/sec CNT100;
   1:  PR[91,1] = PR[90,1] + -1.677;
   1:  PR[91,2] = PR[90,2] + -5.133;
   1:  PR[91,3] = PR[90,3] + 14.616;
   1:L PR[91] R[100]mm/sec CNT100;
   1:  PR[91,1] = PR[90,1] + -1.414;
   1:  PR[91,2] = PR[90,2] + -4.967;
   1:  PR[91,3] = PR[90,3] + 14.620;
   1:L PR[91] R[100]mm/sec CNT100;
   1:  PR[91,1] = PR[90,1] + -1.041;
   1:  PR[91,2] = PR[90,2] + -4.794;
   1:  PR[91,3] = PR[90,3] + 14.622;
   1:L PR[91] R[100]mm/sec CNT100;
   1:  PR[91,1] = PR[90,1] + -0.652;
   1:  PR[91,2] = PR[90,2] + -4.681;
   1:  PR[91,3] = PR[90,3] + 14.624;
   1:L PR[91] R[100]mm/sec CNT100;
   1:  PR[91,1] = PR[90,1] + -0.444;
   1:  PR[91,2] = PR[90,2] + -4.647;
   1:  PR[91,3] = PR[90,3] + 14.627;
   1:L PR[91] R[100]mm/sec CNT100;
   1:  PR[91,1] = PR[90,1] + -0.211;
   1:  PR[91,2] = PR[90,2] + -4.627;
   1:  PR[91,3] = PR[90,3] + 14.628;
   1:L PR[91] R[100]mm/sec CNT100;
   1:  PR[91] = PR[90];
   1:  PR[91,1] = PR[90,1] + 0.141;
   1:  PR[91,2] = PR[90,2] + -5.659;
   1:  PR[91,3] = PR[90,3] + 15.960;
   1:L PR[91] R[100]mm/sec CNT100;
   1:  PR[91,1] = PR[90,1] + 0.562;
   1:  PR[91,2] = PR[90,2] + -5.737;
   1:  PR[91,3] = PR[90,3] + 14.633;
   1:L PR[91] R[100]mm/sec CNT100;
   1:  PR[91,1] = PR[90,1] + 0.899;
   1:  PR[91,2] = PR[90,2] + -5.853;
   1:  PR[91,3] = PR[90,3] + 14.636;
   1:L PR[91] R[100]mm/sec CNT100;
   1:  PR[91,1] = PR[90,1] + 1.298;
   1:  PR[91,2] = PR[90,2] + -6.057;
   1:  PR[91,3] = PR[90,3] + 14.639;
   1:L PR[91] R[100]mm/sec CNT100;
   1:  PR[91,1] = PR[90,1] + 1.678;
   1:  PR[91,2] = PR[90,2] + -6.334;
   1:  PR[91,3] = PR[90,3] + 14.642;
   1:L PR[91] R[100]mm/sec CNT100;
   1:  PR[91,1] = PR[90,1] + 1.994;
   1:  PR[91,2] = PR[90,2] + -6.641;
   1:  PR[91,3] = PR[90,3] + 14.645;
   1:L PR[91] R[100]mm/sec CNT100;
   1:  PR[91,1] = PR[90,1] + 2.314;
   1:  PR[91,2] = PR[90,2] + -7.058;
   1:  PR[91,3] = PR[90,3] + 14.648;
   1:L PR[91] R[100]mm/sec CNT100;
   1:  PR[91,1] = PR[90,1] + 2.884;
   1:  PR[91,2] = PR[90,2] + -8.045;
   1:  PR[91,3] = PR[90,3] + 14.651;
   1:L PR[91] R[100]mm/sec CNT100;
   1:  PR[91,1] = PR[90,1] + 3.316;
   1:  PR[91,2] = PR[90,2] + -8.731;
   1:  PR[91,3] = PR[90,3] + 14.659;
   1:L PR[91] R[100]mm/sec CNT100;
   1:  PR[91,1] = PR[90,1] + 3.595;
   1:  PR[91,2] = PR[90,2] + -9.145;
   1:  PR[91,3] = PR[90,3] + 14.664;
   1:L PR[91] R[100]mm/sec CNT100;
   1:  PR[91,1] = PR[90,1] + 4.131;
   1:  PR[91,2] = PR[90,2] + -9.866;
   1:  PR[91,3] = PR[90,3] + 14.668;
   1:L PR[91] R[100]mm/sec CNT100;
   1:  PR[91,1] = PR[90,1] + 4.771;
   1:  PR[91,2] = PR[90,2] + -10.633;
   1:  PR[91,3] = PR[90,3] + 14.674;
   1:L PR[91] R[100]mm/sec CNT100;
   1:  PR[91,1] = PR[90,1] + 5.313;
   1:  PR[91,2] = PR[90,2] + -11.221;
   1:  PR[91,3] = PR[90,3] + 14.680;
   1:L PR[91] R[100]mm/sec CNT100;
   1:  PR[91,1] = PR[90,1] + 5.951;
   1:  PR[91,2] = PR[90,2] + -11.849;
   1:  PR[91,3] = PR[90,3] + 14.686;
   1:L PR[91] R[100]mm/sec CNT100;
   1:  PR[91,1] = PR[90,1] + 6.621;
   1:  PR[91,2] = PR[90,2] + -12.441;
   1:  PR[91,3] = PR[90,3] + 14.691;
   1:L PR[91] R[100]mm/sec CNT100;
   1:  PR[91,1] = PR[90,1] + 7.322;
   1:  PR[91,2] = PR[90,2] + -13.001;
   1:  PR[91,3] = PR[90,3] + 14.697;
   1:L PR[91] R[100]mm/sec CNT100;
   1:  PR[91,1] = PR[90,1] + 7.683;
   1:  PR[91,2] = PR[90,2] + -13.263;
   1:  PR[91,3] = PR[90,3] + 14.703;
   1:L PR[91] R[100]mm/sec CNT100;
   1:  PR[91,1] = PR[90,1] + 8.046;
   1:  PR[91,2] = PR[90,2] + -13.521;
   1:  PR[91,3] = PR[90,3] + 14.706;
   1:L PR[91] R[100]mm/sec CNT100;
   1:  PR[91,1] = PR[90,1] + 8.800;
   1:  PR[91,2] = PR[90,2] + -14.007;
   1:  PR[91,3] = PR[90,3] + 14.709;
   1:L PR[91] R[100]mm/sec CNT100;
   1:  PR[91,1] = PR[90,1] + 9.576;
   1:  PR[91,2] = PR[90,2] + -14.455;
   1:  PR[91,3] = PR[90,3] + 14.715;
   1:L PR[91] R[100]mm/sec CNT100;
   1:  PR[91,1] = PR[90,1] + 10.375;
   1:  PR[91,2] = PR[90,2] + -14.865;
   1:  PR[91,3] = PR[90,3] + 14.721;
   1:L PR[91] R[100]mm/sec CNT100;
   1:  PR[91,1] = PR[90,1] + 11.098;
   1:  PR[91,2] = PR[90,2] + -15.196;
   1:  PR[91,3] = PR[90,3] + 14.727;
   1:L PR[91] R[100]mm/sec CNT100;
   1:  PR[91,1] = PR[90,1] + 12.093;
   1:  PR[91,2] = PR[90,2] + -15.593;
   1:  PR[91,3] = PR[90,3] + 14.733;
   1:L PR[91] R[100]mm/sec CNT100;
   1:  PR[91,1] = PR[90,1] + 12.613;
   1:  PR[91,2] = PR[90,2] + -15.773;
   1:  PR[91,3] = PR[90,3] + 14.740;
   1:L PR[91] R[100]mm/sec CNT100;
   1:  PR[91,1] = PR[90,1] + 13.395;
   1:  PR[91,2] = PR[90,2] + -16.014;
   1:  PR[91,3] = PR[90,3] + 14.743;
   1:L PR[91] R[100]mm/sec CNT100;
   1:  PR[91,1] = PR[90,1] + 14.188;
   1:  PR[91,2] = PR[90,2] + -16.220;
   1:  PR[91,3] = PR[90,3] + 14.749;
   1:L PR[91] R[100]mm/sec CNT100;
   1:  PR[91,1] = PR[90,1] + 14.993;
   1:  PR[91,2] = PR[90,2] + -16.391;
   1:  PR[91,3] = PR[90,3] + 14.754;
   1:L PR[91] R[100]mm/sec CNT100;
   1:  PR[91,1] = PR[90,1] + 15.807;
   1:  PR[91,2] = PR[90,2] + -16.527;
   1:  PR[91,3] = PR[90,3] + 14.760;
   1:L PR[91] R[100]mm/sec CNT100;
   1:  PR[91,1] = PR[90,1] + 16.653;
   1:  PR[91,2] = PR[90,2] + -16.628;
   1:  PR[91,3] = PR[90,3] + 14.765;
   1:L PR[91] R[100]mm/sec CNT100;
   1:  PR[91,1] = PR[90,1] + 17.544;
   1:  PR[91,2] = PR[90,2] + -16.692;
   1:  PR[91,3] = PR[90,3] + 14.771;
   1:L PR[91] R[100]mm/sec CNT100;
   1:  PR[91,1] = PR[90,1] + 18.186;
   1:  PR[91,2] = PR[90,2] + -16.708;
   1:  PR[91,3] = PR[90,3] + 14.777;
   1:L PR[91] R[100]mm/sec CNT100;
   1:  PR[91,1] = PR[90,1] + 19.324;
   1:  PR[91,2] = PR[90,2] + -16.690;
   1:  PR[91,3] = PR[90,3] + 14.781;
   1:L PR[91] R[100]mm/sec CNT100;
   1:  PR[91,1] = PR[90,1] + 20.205;
   1:  PR[91,2] = PR[90,2] + -16.624;
   1:  PR[91,3] = PR[90,3] + 14.789;
   1:L PR[91] R[100]mm/sec CNT100;
   1:  PR[91,1] = PR[90,1] + 21.081;
   1:  PR[91,2] = PR[90,2] + -16.516;
   1:  PR[91,3] = PR[90,3] + 14.795;
   1:L PR[91] R[100]mm/sec CNT100;
   1:  PR[91,1] = PR[90,1] + 21.950;
   1:  PR[91,2] = PR[90,2] + -16.365;
   1:  PR[91,3] = PR[90,3] + 14.800;
   1:L PR[91] R[100]mm/sec CNT100;
   1:  PR[91,1] = PR[90,1] + 22.807;
   1:  PR[91,2] = PR[90,2] + -16.173;
   1:  PR[91,3] = PR[90,3] + 14.806;
   1:L PR[91] R[100]mm/sec CNT100;
   1:  PR[91,1] = PR[90,1] + 23.651;
   1:  PR[91,2] = PR[90,2] + -15.941;
   1:  PR[91,3] = PR[90,3] + 14.812;
   1:L PR[91] R[100]mm/sec CNT100;
   1:  PR[91,1] = PR[90,1] + 24.477;
   1:  PR[91,2] = PR[90,2] + -15.669;
   1:  PR[91,3] = PR[90,3] + 14.818;
   1:L PR[91] R[100]mm/sec CNT100;
   1:  PR[91,1] = PR[90,1] + 25.287;
   1:  PR[91,2] = PR[90,2] + -15.359;
   1:  PR[91,3] = PR[90,3] + 14.824;
   1:L PR[91] R[100]mm/sec CNT100;
   1:  PR[91,1] = PR[90,1] + 26.079;
   1:  PR[91,2] = PR[90,2] + -15.011;
   1:  PR[91,3] = PR[90,3] + 14.830;
   1:L PR[91] R[100]mm/sec CNT100;
   1:  PR[91,1] = PR[90,1] + 26.851;
   1:  PR[91,2] = PR[90,2] + -14.626;
   1:  PR[91,3] = PR[90,3] + 14.835;
   1:L PR[91] R[100]mm/sec CNT100;
   1:  PR[91,1] = PR[90,1] + 27.601;
   1:  PR[91,2] = PR[90,2] + -14.205;
   1:  PR[91,3] = PR[90,3] + 14.841;
   1:L PR[91] R[100]mm/sec CNT100;
   1:  PR[91,1] = PR[90,1] + 28.328;
   1:  PR[91,2] = PR[90,2] + -13.750;
   1:  PR[91,3] = PR[90,3] + 14.847;
   1:L PR[91] R[100]mm/sec CNT100;
   1:  PR[91,1] = PR[90,1] + 29.029;
   1:  PR[91,2] = PR[90,2] + -13.261;
   1:  PR[91,3] = PR[90,3] + 14.852;
   1:L PR[91] R[100]mm/sec CNT100;
   1:  PR[91,1] = PR[90,1] + 29.705;
   1:  PR[91,2] = PR[90,2] + -12.740;
   1:  PR[91,3] = PR[90,3] + 14.858;
   1:L PR[91] R[100]mm/sec CNT100;
   1:  PR[91,1] = PR[90,1] + 30.352;
   1:  PR[91,2] = PR[90,2] + -12.187;
   1:  PR[91,3] = PR[90,3] + 14.864;
   1:L PR[91] R[100]mm/sec CNT100;
   1:  PR[91,1] = PR[90,1] + 30.969;
   1:  PR[91,2] = PR[90,2] + -11.605;
   1:  PR[91,3] = PR[90,3] + 14.869;
   1:L PR[91] R[100]mm/sec CNT100;
   1:  PR[91,1] = PR[90,1] + 31.557;
   1:  PR[91,2] = PR[90,2] + -10.993;
   1:  PR[91,3] = PR[90,3] + 14.875;
   1:L PR[91] R[100]mm/sec CNT100;
   1:  PR[91,1] = PR[90,1] + 32.112;
   1:  PR[91,2] = PR[90,2] + -10.353;
   1:  PR[91,3] = PR[90,3] + 14.881;
   1:L PR[91] R[100]mm/sec CNT100;
   1:  PR[91,1] = PR[90,1] + 32.637;
   1:  PR[91,2] = PR[90,2] + -9.684;
   1:  PR[91,3] = PR[90,3] + 14.886;
   1:L PR[91] R[100]mm/sec CNT100;
   1:  PR[91,1] = PR[90,1] + 33.121;
   1:  PR[91,2] = PR[90,2] + -8.999;
   1:  PR[91,3] = PR[90,3] + 14.892;
   1:L PR[91] R[100]mm/sec CNT100;
   1:  PR[91,1] = PR[90,1] + 33.572;
   1:  PR[91,2] = PR[90,2] + -8.288;
   1:  PR[91,3] = PR[90,3] + 14.898;
   1:L PR[91] R[100]mm/sec CNT100;
   1:  PR[91,1] = PR[90,1] + 33.989;
   1:  PR[91,2] = PR[90,2] + -7.558;
   1:  PR[91,3] = PR[90,3] + 14.903;
   1:L PR[91] R[100]mm/sec CNT100;
   1:  PR[91,1] = PR[90,1] + 34.368;
   1:  PR[91,2] = PR[90,2] + -6.812;
   1:  PR[91,3] = PR[90,3] + 14.909;
   1:L PR[91] R[100]mm/sec CNT100;
   1:  PR[91,1] = PR[90,1] + 34.709;
   1:  PR[91,2] = PR[90,2] + -6.052;
   1:  PR[91,3] = PR[90,3] + 14.914;
   1:L PR[91] R[100]mm/sec CNT100;
   1:  PR[91,1] = PR[90,1] + 35.012;
   1:  PR[91,2] = PR[90,2] + -5.283;
   1:  PR[91,3] = PR[90,3] + 14.920;
   1:L PR[91] R[100]mm/sec CNT100;
   1:  PR[91,1] = PR[90,1] + 35.275;
   1:  PR[91,2] = PR[90,2] + -4.503;
   1:  PR[91,3] = PR[90,3] + 14.925;
   1:L PR[91] R[100]mm/sec CNT100;
   1:  PR[91,1] = PR[90,1] + 35.499;
   1:  PR[91,2] = PR[90,2] + -3.714;
   1:  PR[91,3] = PR[90,3] + 14.931;
   1:L PR[91] R[100]mm/sec CNT100;
   1:  PR[91,1] = PR[90,1] + 35.683;
   1:  PR[91,2] = PR[90,2] + -2.913;
   1:  PR[91,3] = PR[90,3] + 14.936;
   1:L PR[91] R[100]mm/sec CNT100;
   1:  PR[91,1] = PR[90,1] + 35.826;
   1:  PR[91,2] = PR[90,2] + -2.101;
   1:  PR[91,3] = PR[90,3] + 14.942;
   1:L PR[91] R[100]mm/sec CNT100;
   1:  PR[91,1] = PR[90,1] + 35.928;
   1:  PR[91,2] = PR[90,2] + -1.274;
   1:  PR[91,3] = PR[90,3] + 14.947;
   1:L PR[91] R[100]mm/sec CNT100;
   1:  PR[91,1] = PR[90,1] + 35.990;
   1:  PR[91,2] = PR[90,2] + -0.432;
   1:  PR[91,3] = PR[90,3] + 14.953;
   1:L PR[91] R[100]mm/sec CNT100;
   1:  PR[91,1] = PR[90,1] + 36.011;
   1:  PR[91,2] = PR[90,2] + 0.428;
   1:  PR[91,3] = PR[90,3] + 14.959;
   1:L PR[91] R[100]mm/sec CNT100;
   1:  PR[91,1] = PR[90,1] + 35.990;
   1:  PR[91,2] = PR[90,2] + 1.287;
   1:  PR[91,3] = PR[90,3] + 14.964;
   1:L PR[91] R[100]mm/sec CNT100;
   1:  PR[91,1] = PR[90,1] + 35.928;
   1:  PR[91,2] = PR[90,2] + 2.129;
   1:  PR[91,3] = PR[90,3] + 14.970;
   1:L PR[91] R[100]mm/sec CNT100;
   1:  PR[91,1] = PR[90,1] + 35.826;
   1:  PR[91,2] = PR[90,2] + 2.956;
   1:  PR[91,3] = PR[90,3] + 14.976;
   1:L PR[91] R[100]mm/sec CNT100;
   1:  PR[91,1] = PR[90,1] + 35.683;
   1:  PR[91,2] = PR[90,2] + 3.769;
   1:  PR[91,3] = PR[90,3] + 14.981;
   1:L PR[91] R[100]mm/sec CNT100;
   1:  PR[91,1] = PR[90,1] + 35.499;
   1:  PR[91,2] = PR[90,2] + 4.569;
   1:  PR[91,3] = PR[90,3] + 14.987;
   1:L PR[91] R[100]mm/sec CNT100;
   1:  PR[91,1] = PR[90,1] + 35.275;
   1:  PR[91,2] = PR[90,2] + 5.358;
   1:  PR[91,3] = PR[90,3] + 14.992;
   1:L PR[91] R[100]mm/sec CNT100;
   1:  PR[91,1] = PR[90,1] + 35.012;
   1:  PR[91,2] = PR[90,2] + 6.138;
   1:  PR[91,3] = PR[90,3] + 14.998;
   1:L PR[91] R[100]mm/sec CNT100;
   1:  PR[91,1] = PR[90,1] + 34.709;
   1:  PR[91,2] = PR[90,2] + 6.908;
   1:  PR[91,3] = PR[90,3] + 15.003;
   1:L PR[91] R[100]mm/sec CNT100;
   1:  PR[91,1] = PR[90,1] + 34.368;
   1:  PR[91,2] = PR[90,2] + 7.667;
   1:  PR[91,3] = PR[90,3] + 15.009;
   1:L PR[91] R[100]mm/sec CNT100;
   1:  PR[91,1] = PR[90,1] + 33.989;
   1:  PR[91,2] = PR[90,2] + 8.413;
   1:  PR[91,3] = PR[90,3] + 15.014;
   1:L PR[91] R[100]mm/sec CNT100;
   1:  PR[91,1] = PR[90,1] + 33.572;
   1:  PR[91,2] = PR[90,2] + 9.143;
   1:  PR[91,3] = PR[90,3] + 15.020;
   1:L PR[91] R[100]mm/sec CNT100;
   1:  PR[91,1] = PR[90,1] + 33.121;
   1:  PR[91,2] = PR[90,2] + 9.854;
   1:  PR[91,3] = PR[90,3] + 15.025;
   1:L PR[91] R[100]mm/sec CNT100;
   1:  PR[91,1] = PR[90,1] + 32.634;
   1:  PR[91,2] = PR[90,2] + 10.543;
   1:  PR[91,3] = PR[90,3] + 15.031;
   1:L PR[91] R[100]mm/sec CNT100;
   1:  PR[91,1] = PR[90,1] + 32.112;
   1:  PR[91,2] = PR[90,2] + 11.209;
   1:  PR[91,3] = PR[90,3] + 15.036;
   1:L PR[91] R[100]mm/sec CNT100;
   1:  PR[91,1] = PR[90,1] + 31.557;
   1:  PR[91,2] = PR[90,2] + 11.848;
   1:  PR[91,3] = PR[90,3] + 15.042;
   1:L PR[91] R[100]mm/sec CNT100;
   1:  PR[91,1] = PR[90,1] + 30.969;
   1:  PR[91,2] = PR[90,2] + 12.460;
   1:  PR[91,3] = PR[90,3] + 15.048;
   1:L PR[91] R[100]mm/sec CNT100;
   1:  PR[91,1] = PR[90,1] + 30.352;
   1:  PR[91,2] = PR[90,2] + 13.043;
   1:  PR[91,3] = PR[90,3] + 15.053;
   1:L PR[91] R[100]mm/sec CNT100;
   1:  PR[91,1] = PR[90,1] + 29.705;
   1:  PR[91,2] = PR[90,2] + 13.595;
   1:  PR[91,3] = PR[90,3] + 15.059;
   1:L PR[91] R[100]mm/sec CNT100;
   1:  PR[91,1] = PR[90,1] + 29.029;
   1:  PR[91,2] = PR[90,2] + 14.117;
   1:  PR[91,3] = PR[90,3] + 15.065;
   1:L PR[91] R[100]mm/sec CNT100;
   1:  PR[91,1] = PR[90,1] + 28.622;
   1:  PR[91,2] = PR[90,2] + 14.402;
   1:  PR[91,3] = PR[90,3] + 15.070;
   1:L PR[91] R[100]mm/sec CNT100;
   1:  PR[91,1] = PR[90,1] + 28.329;
   1:  PR[91,2] = PR[90,2] + 14.605;
   1:  PR[91,3] = PR[90,3] + 15.074;
   1:L PR[91] R[100]mm/sec CNT100;
   1:  PR[91,1] = PR[90,1] + 27.601;
   1:  PR[91,2] = PR[90,2] + 15.060;
   1:  PR[91,3] = PR[90,3] + 15.076;
   1:L PR[91] R[100]mm/sec CNT100;
   1:  PR[91,1] = PR[90,1] + 26.850;
   1:  PR[91,2] = PR[90,2] + 15.481;
   1:  PR[91,3] = PR[90,3] + 15.082;
   1:L PR[91] R[100]mm/sec CNT100;
   1:  PR[91,1] = PR[90,1] + 26.585;
   1:  PR[91,2] = PR[90,2] + 15.615;
   1:  PR[91,3] = PR[90,3] + 15.088;
   1:L PR[91] R[100]mm/sec CNT100;
   1:  PR[91,1] = PR[90,1] + 26.080;
   1:  PR[91,2] = PR[90,2] + 15.866;
   1:  PR[91,3] = PR[90,3] + 15.089;
   1:L PR[91] R[100]mm/sec CNT100;
   1:  PR[91,1] = PR[90,1] + 25.287;
   1:  PR[91,2] = PR[90,2] + 16.214;
   1:  PR[91,3] = PR[90,3] + 15.093;
   1:L PR[91] R[100]mm/sec CNT100;
   1:  PR[91,1] = PR[90,1] + 24.478;
   1:  PR[91,2] = PR[90,2] + 16.524;
   1:  PR[91,3] = PR[90,3] + 15.099;
   1:L PR[91] R[100]mm/sec CNT100;
   1:  PR[91,1] = PR[90,1] + 23.632;
   1:  PR[91,2] = PR[90,2] + 16.801;
   1:  PR[91,3] = PR[90,3] + 15.105;
   1:L PR[91] R[100]mm/sec CNT100;
   1:  PR[91,1] = PR[90,1] + 22.807;
   1:  PR[91,2] = PR[90,2] + 17.028;
   1:  PR[91,3] = PR[90,3] + 15.111;
   1:L PR[91] R[100]mm/sec CNT100;
   1:  PR[91,1] = PR[90,1] + 21.949;
   1:  PR[91,2] = PR[90,2] + 17.220;
   1:  PR[91,3] = PR[90,3] + 15.116;
   1:L PR[91] R[100]mm/sec CNT100;
   1:  PR[91,1] = PR[90,1] + 21.081;
   1:  PR[91,2] = PR[90,2] + 17.371;
   1:  PR[91,3] = PR[90,3] + 15.122;
   1:L PR[91] R[100]mm/sec CNT100;
   1:  PR[91,1] = PR[90,1] + 20.204;
   1:  PR[91,2] = PR[90,2] + 17.479;
   1:  PR[91,3] = PR[90,3] + 15.128;
   1:L PR[91] R[100]mm/sec CNT100;
   1:  PR[91,1] = PR[90,1] + 19.768;
   1:  PR[91,2] = PR[90,2] + 17.513;
   1:  PR[91,3] = PR[90,3] + 15.134;
   1:L PR[91] R[100]mm/sec CNT100;
   1:  PR[91,1] = PR[90,1] + 19.323;
   1:  PR[91,2] = PR[90,2] + 17.545;
   1:  PR[91,3] = PR[90,3] + 15.137;
   1:L PR[91] R[100]mm/sec CNT100;
   1:  PR[91,1] = PR[90,1] + 18.434;
   1:  PR[91,2] = PR[90,2] + 17.568;
   1:  PR[91,3] = PR[90,3] + 15.140;
   1:L PR[91] R[100]mm/sec CNT100;
   1:  PR[91,1] = PR[90,1] + 17.544;
   1:  PR[91,2] = PR[90,2] + 17.547;
   1:  PR[91,3] = PR[90,3] + 15.146;
   1:L PR[91] R[100]mm/sec CNT100;
   1:  PR[91,1] = PR[90,1] + 16.653;
   1:  PR[91,2] = PR[90,2] + 17.483;
   1:  PR[91,3] = PR[90,3] + 15.152;
   1:L PR[91] R[100]mm/sec CNT100;
   1:  PR[91,1] = PR[90,1] + 15.807;
   1:  PR[91,2] = PR[90,2] + 17.382;
   1:  PR[91,3] = PR[90,3] + 15.158;
   1:L PR[91] R[100]mm/sec CNT100;
   1:  PR[91,1] = PR[90,1] + 14.995;
   1:  PR[91,2] = PR[90,2] + 17.247;
   1:  PR[91,3] = PR[90,3] + 15.163;
   1:L PR[91] R[100]mm/sec CNT100;
   1:  PR[91,1] = PR[90,1] + 13.877;
   1:  PR[91,2] = PR[90,2] + 16.999;
   1:  PR[91,3] = PR[90,3] + 15.169;
   1:L PR[91] R[100]mm/sec CNT100;
   1:  PR[91,1] = PR[90,1] + 13.397;
   1:  PR[91,2] = PR[90,2] + 16.870;
   1:  PR[91,3] = PR[90,3] + 15.176;
   1:L PR[91] R[100]mm/sec CNT100;
   1:  PR[91,1] = PR[90,1] + 12.615;
   1:  PR[91,2] = PR[90,2] + 16.629;
   1:  PR[91,3] = PR[90,3] + 15.180;
   1:L PR[91] R[100]mm/sec CNT100;
   1:  PR[91,1] = PR[90,1] + 11.849;
   1:  PR[91,2] = PR[90,2] + 16.356;
   1:  PR[91,3] = PR[90,3] + 15.185;
   1:L PR[91] R[100]mm/sec CNT100;
   1:  PR[91,1] = PR[90,1] + 11.100;
   1:  PR[91,2] = PR[90,2] + 16.052;
   1:  PR[91,3] = PR[90,3] + 15.191;
   1:L PR[91] R[100]mm/sec CNT100;
   1:  PR[91,1] = PR[90,1] + 10.368;
   1:  PR[91,2] = PR[90,2] + 15.717;
   1:  PR[91,3] = PR[90,3] + 15.196;
   1:L PR[91] R[100]mm/sec CNT100;
   1:  PR[91,1] = PR[90,1] + 9.575;
   1:  PR[91,2] = PR[90,2] + 15.310;
   1:  PR[91,3] = PR[90,3] + 15.201;
   1:L PR[91] R[100]mm/sec CNT100;
   1:  PR[91,1] = PR[90,1] + 8.800;
   1:  PR[91,2] = PR[90,2] + 14.862;
   1:  PR[91,3] = PR[90,3] + 15.207;
   1:L PR[91] R[100]mm/sec CNT100;
   1:  PR[91,1] = PR[90,1] + 8.046;
   1:  PR[91,2] = PR[90,2] + 14.376;
   1:  PR[91,3] = PR[90,3] + 15.213;
   1:L PR[91] R[100]mm/sec CNT100;
   1:  PR[91,1] = PR[90,1] + 7.683;
   1:  PR[91,2] = PR[90,2] + 14.119;
   1:  PR[91,3] = PR[90,3] + 15.219;
   1:L PR[91] R[100]mm/sec CNT100;
   1:  PR[91,1] = PR[90,1] + 7.322;
   1:  PR[91,2] = PR[90,2] + 13.856;
   1:  PR[91,3] = PR[90,3] + 15.222;
   1:L PR[91] R[100]mm/sec CNT100;
   1:  PR[91,1] = PR[90,1] + 6.621;
   1:  PR[91,2] = PR[90,2] + 13.297;
   1:  PR[91,3] = PR[90,3] + 15.225;
   1:L PR[91] R[100]mm/sec CNT100;
   1:  PR[91,1] = PR[90,1] + 5.951;
   1:  PR[91,2] = PR[90,2] + 12.704;
   1:  PR[91,3] = PR[90,3] + 15.231;
   1:L PR[91] R[100]mm/sec CNT100;
   1:  PR[91,1] = PR[90,1] + 5.308;
   1:  PR[91,2] = PR[90,2] + 12.071;
   1:  PR[91,3] = PR[90,3] + 15.237;
   1:L PR[91] R[100]mm/sec CNT100;
   1:  PR[91,1] = PR[90,1] + 4.705;
   1:  PR[91,2] = PR[90,2] + 11.415;
   1:  PR[91,3] = PR[90,3] + 15.243;
   1:L PR[91] R[100]mm/sec CNT100;
   1:  PR[91,1] = PR[90,1] + 4.132;
   1:  PR[91,2] = PR[90,2] + 10.722;
   1:  PR[91,3] = PR[90,3] + 15.249;
   1:L PR[91] R[100]mm/sec CNT100;
   1:  PR[91,1] = PR[90,1] + 3.595;
   1:  PR[91,2] = PR[90,2] + 10.000;
   1:  PR[91,3] = PR[90,3] + 15.255;
   1:L PR[91] R[100]mm/sec CNT100;
   1:  PR[91,1] = PR[90,1] + 3.316;
   1:  PR[91,2] = PR[90,2] + 9.587;
   1:  PR[91,3] = PR[90,3] + 15.261;
   1:L PR[91] R[100]mm/sec CNT100;
   1:  PR[91,1] = PR[90,1] + 2.884;
   1:  PR[91,2] = PR[90,2] + 8.901;
   1:  PR[91,3] = PR[90,3] + 15.264;
   1:L PR[91] R[100]mm/sec CNT100;
   1:  PR[91,1] = PR[90,1] + 2.313;
   1:  PR[91,2] = PR[90,2] + 7.910;
   1:  PR[91,3] = PR[90,3] + 15.270;
   1:L PR[91] R[100]mm/sec CNT100;
   1:  PR[91,1] = PR[90,1] + 1.993;
   1:  PR[91,2] = PR[90,2] + 7.495;
   1:  PR[91,3] = PR[90,3] + 15.277;
   1:L PR[91] R[100]mm/sec CNT100;
   1:  PR[91,1] = PR[90,1] + 1.672;
   1:  PR[91,2] = PR[90,2] + 7.184;
   1:  PR[91,3] = PR[90,3] + 15.281;
   1:L PR[91] R[100]mm/sec CNT100;
   1:  PR[91,1] = PR[90,1] + 1.338;
   1:  PR[91,2] = PR[90,2] + 6.937;
   1:  PR[91,3] = PR[90,3] + 15.284;
   1:L PR[91] R[100]mm/sec CNT100;
   1:  PR[91,1] = PR[90,1] + 0.960;
   1:  PR[91,2] = PR[90,2] + 6.733;
   1:  PR[91,3] = PR[90,3] + 15.287;
   1:L PR[91] R[100]mm/sec CNT100;
   1:  PR[91,1] = PR[90,1] + 0.479;
   1:  PR[91,2] = PR[90,2] + 6.572;
   1:  PR[91,3] = PR[90,3] + 15.289;
   1:L PR[91] R[100]mm/sec CNT100;
   1:  PR[91,1] = PR[90,1] + 0.142;
   1:  PR[91,2] = PR[90,2] + 6.515;
   1:  PR[91,3] = PR[90,3] + 15.293;
   1:L PR[91] R[100]mm/sec CNT100;
   1:  PR[91,1] = PR[90,1] + -0.288;
   1:  PR[91,2] = PR[90,2] + 6.507;
   1:  PR[91,3] = PR[90,3] + 15.295;
   1:L PR[91] R[100]mm/sec CNT100;
   1:  PR[91,1] = PR[90,1] + -0.804;
   1:  PR[91,2] = PR[90,2] + 6.593;
   1:  PR[91,3] = PR[90,3] + 15.298;
   1:L PR[91] R[100]mm/sec CNT100;
   1:  PR[91,1] = PR[90,1] + -1.209;
   1:  PR[91,2] = PR[90,2] + 6.739;
   1:  PR[91,3] = PR[90,3] + 15.301;
   1:L PR[91] R[100]mm/sec CNT100;
   1:  PR[91,1] = PR[90,1] + -1.582;
   1:  PR[91,2] = PR[90,2] + 6.941;
   1:  PR[91,3] = PR[90,3] + 15.304;
   1:L PR[91] R[100]mm/sec CNT100;
   1:  PR[91,1] = PR[90,1] + -1.923;
   1:  PR[91,2] = PR[90,2] + 7.195;
   1:  PR[91,3] = PR[90,3] + 15.307;
   1:L PR[91] R[100]mm/sec CNT100;
   1:  PR[91,1] = PR[90,1] + -2.236;
   1:  PR[91,2] = PR[90,2] + 7.501;
   1:  PR[91,3] = PR[90,3] + 15.310;
   1:L PR[91] R[100]mm/sec CNT100;
   1:  PR[91,1] = PR[90,1] + -2.554;
   1:  PR[91,2] = PR[90,2] + 7.917;
   1:  PR[91,3] = PR[90,3] + 15.313;
   1:L PR[91] R[100]mm/sec CNT100;
   1:  PR[91,1] = PR[90,1] + -3.124;
   1:  PR[91,2] = PR[90,2] + 8.910;
   1:  PR[91,3] = PR[90,3] + 15.316;
   1:L PR[91] R[100]mm/sec CNT100;
   1:  PR[91,1] = PR[90,1] + -3.556;
   1:  PR[91,2] = PR[90,2] + 9.598;
   1:  PR[91,3] = PR[90,3] + 15.324;
   1:L PR[91] R[100]mm/sec CNT100;
   1:  PR[91,1] = PR[90,1] + -3.835;
   1:  PR[91,2] = PR[90,2] + 10.011;
   1:  PR[91,3] = PR[90,3] + 15.329;
   1:L PR[91] R[100]mm/sec CNT100;
   1:  PR[91,1] = PR[90,1] + -4.371;
   1:  PR[91,2] = PR[90,2] + 10.731;
   1:  PR[91,3] = PR[90,3] + 15.333;
   1:L PR[91] R[100]mm/sec CNT100;
   1:  PR[91,1] = PR[90,1] + -5.011;
   1:  PR[91,2] = PR[90,2] + 11.495;
   1:  PR[91,3] = PR[90,3] + 15.339;
   1:L PR[91] R[100]mm/sec CNT100;
   1:  PR[91,1] = PR[90,1] + -5.553;
   1:  PR[91,2] = PR[90,2] + 12.080;
   1:  PR[91,3] = PR[90,3] + 15.345;
   1:L PR[91] R[100]mm/sec CNT100;
   1:  PR[91,1] = PR[90,1] + -6.192;
   1:  PR[91,2] = PR[90,2] + 12.706;
   1:  PR[91,3] = PR[90,3] + 15.351;
   1:L PR[91] R[100]mm/sec CNT100;
   1:  PR[91,1] = PR[90,1] + -6.864;
   1:  PR[91,2] = PR[90,2] + 13.298;
   1:  PR[91,3] = PR[90,3] + 15.356;
   1:L PR[91] R[100]mm/sec CNT100;
   1:  PR[91,1] = PR[90,1] + -7.302;
   1:  PR[91,2] = PR[90,2] + 13.650;
   1:  PR[91,3] = PR[90,3] + 15.362;
   1:L PR[91] R[100]mm/sec CNT100;
   1:  PR[91,1] = PR[90,1] + -7.561;
   1:  PR[91,2] = PR[90,2] + 13.854;
   1:  PR[91,3] = PR[90,3] + 15.366;
   1:L PR[91] R[100]mm/sec CNT100;
   1:  PR[91,1] = PR[90,1] + -8.288;
   1:  PR[91,2] = PR[90,2] + 14.376;
   1:  PR[91,3] = PR[90,3] + 15.368;
   1:L PR[91] R[100]mm/sec CNT100;
   1:  PR[91,1] = PR[90,1] + -9.237;
   1:  PR[91,2] = PR[90,2] + 14.977;
   1:  PR[91,3] = PR[90,3] + 15.374;
   1:L PR[91] R[100]mm/sec CNT100;
   1:  PR[91,1] = PR[90,1] + -9.819;
   1:  PR[91,2] = PR[90,2] + 15.311;
   1:  PR[91,3] = PR[90,3] + 15.382;
   1:L PR[91] R[100]mm/sec CNT100;
   1:  PR[91,1] = PR[90,1] + -10.621;
   1:  PR[91,2] = PR[90,2] + 15.723;
   1:  PR[91,3] = PR[90,3] + 15.386;
   1:L PR[91] R[100]mm/sec CNT100;
   1:  PR[91,1] = PR[90,1] + -11.344;
   1:  PR[91,2] = PR[90,2] + 16.055;
   1:  PR[91,3] = PR[90,3] + 15.392;
   1:L PR[91] R[100]mm/sec CNT100;
   1:  PR[91,1] = PR[90,1] + -12.091;
   1:  PR[91,2] = PR[90,2] + 16.359;
   1:  PR[91,3] = PR[90,3] + 15.398;
   1:L PR[91] R[100]mm/sec CNT100;
   1:  PR[91,1] = PR[90,1] + -13.222;
   1:  PR[91,2] = PR[90,2] + 16.749;
   1:  PR[91,3] = PR[90,3] + 15.403;
   1:L PR[91] R[100]mm/sec CNT100;
   1:  PR[91,1] = PR[90,1] + -14.436;
   1:  PR[91,2] = PR[90,2] + 17.078;
   1:  PR[91,3] = PR[90,3] + 15.411;
   1:L PR[91] R[100]mm/sec CNT100;
   1:  PR[91,1] = PR[90,1] + -15.238;
   1:  PR[91,2] = PR[90,2] + 17.248;
   1:  PR[91,3] = PR[90,3] + 15.419;
   1:L PR[91] R[100]mm/sec CNT100;
   1:  PR[91,1] = PR[90,1] + -15.977;
   1:  PR[91,2] = PR[90,2] + 17.372;
   1:  PR[91,3] = PR[90,3] + 15.425;
   1:L PR[91] R[100]mm/sec CNT100;
   1:  PR[91,1] = PR[90,1] + -16.899;
   1:  PR[91,2] = PR[90,2] + 17.484;
   1:  PR[91,3] = PR[90,3] + 15.430;
   1:L PR[91] R[100]mm/sec CNT100;
   1:  PR[91,1] = PR[90,1] + -17.789;
   1:  PR[91,2] = PR[90,2] + 17.547;
   1:  PR[91,3] = PR[90,3] + 15.436;
   1:L PR[91] R[100]mm/sec CNT100;
   1:  PR[91,1] = PR[90,1] + -18.679;
   1:  PR[91,2] = PR[90,2] + 17.567;
   1:  PR[91,3] = PR[90,3] + 15.442;
   1:L PR[91] R[100]mm/sec CNT100;
   1:  PR[91,1] = PR[90,1] + -19.567;
   1:  PR[91,2] = PR[90,2] + 17.544;
   1:  PR[91,3] = PR[90,3] + 15.448;
   1:L PR[91] R[100]mm/sec CNT100;
   1:  PR[91,1] = PR[90,1] + -20.011;
   1:  PR[91,2] = PR[90,2] + 17.513;
   1:  PR[91,3] = PR[90,3] + 15.454;
   1:L PR[91] R[100]mm/sec CNT100;
   1:  PR[91,1] = PR[90,1] + -20.448;
   1:  PR[91,2] = PR[90,2] + 17.478;
   1:  PR[91,3] = PR[90,3] + 15.457;
   1:L PR[91] R[100]mm/sec CNT100;
   1:  PR[91,1] = PR[90,1] + -21.326;
   1:  PR[91,2] = PR[90,2] + 17.370;
   1:  PR[91,3] = PR[90,3] + 15.460;
   1:L PR[91] R[100]mm/sec CNT100;
   1:  PR[91,1] = PR[90,1] + -22.194;
   1:  PR[91,2] = PR[90,2] + 17.219;
   1:  PR[91,3] = PR[90,3] + 15.465;
   1:L PR[91] R[100]mm/sec CNT100;
   1:  PR[91,1] = PR[90,1] + -23.051;
   1:  PR[91,2] = PR[90,2] + 17.028;
   1:  PR[91,3] = PR[90,3] + 15.471;
   1:L PR[91] R[100]mm/sec CNT100;
   1:  PR[91,1] = PR[90,1] + -23.895;
   1:  PR[91,2] = PR[90,2] + 16.795;
   1:  PR[91,3] = PR[90,3] + 15.477;
   1:L PR[91] R[100]mm/sec CNT100;
   1:  PR[91,1] = PR[90,1] + -24.721;
   1:  PR[91,2] = PR[90,2] + 16.524;
   1:  PR[91,3] = PR[90,3] + 15.483;
   1:L PR[91] R[100]mm/sec CNT100;
   1:  PR[91,1] = PR[90,1] + -25.530;
   1:  PR[91,2] = PR[90,2] + 16.213;
   1:  PR[91,3] = PR[90,3] + 15.489;
   1:L PR[91] R[100]mm/sec CNT100;
   1:  PR[91,1] = PR[90,1] + -26.321;
   1:  PR[91,2] = PR[90,2] + 15.864;
   1:  PR[91,3] = PR[90,3] + 15.495;
   1:L PR[91] R[100]mm/sec CNT100;
   1:  PR[91,1] = PR[90,1] + -27.093;
   1:  PR[91,2] = PR[90,2] + 15.479;
   1:  PR[91,3] = PR[90,3] + 15.500;
   1:L PR[91] R[100]mm/sec CNT100;
   1:  PR[91,1] = PR[90,1] + -27.843;
   1:  PR[91,2] = PR[90,2] + 15.057;
   1:  PR[91,3] = PR[90,3] + 15.506;
   1:L PR[91] R[100]mm/sec CNT100;
   1:  PR[91,1] = PR[90,1] + -28.570;
   1:  PR[91,2] = PR[90,2] + 14.601;
   1:  PR[91,3] = PR[90,3] + 15.512;
   1:L PR[91] R[100]mm/sec CNT100;
   1:  PR[91,1] = PR[90,1] + -28.864;
   1:  PR[91,2] = PR[90,2] + 14.397;
   1:  PR[91,3] = PR[90,3] + 15.517;
   1:L PR[91] R[100]mm/sec CNT100;
   1:  PR[91,1] = PR[90,1] + -29.270;
   1:  PR[91,2] = PR[90,2] + 14.113;
   1:  PR[91,3] = PR[90,3] + 15.520;
   1:L PR[91] R[100]mm/sec CNT100;
   1:  PR[91,1] = PR[90,1] + -29.946;
   1:  PR[91,2] = PR[90,2] + 13.591;
   1:  PR[91,3] = PR[90,3] + 15.523;
   1:L PR[91] R[100]mm/sec CNT100;
   1:  PR[91,1] = PR[90,1] + -30.593;
   1:  PR[91,2] = PR[90,2] + 13.039;
   1:  PR[91,3] = PR[90,3] + 15.529;
   1:L PR[91] R[100]mm/sec CNT100;
   1:  PR[91,1] = PR[90,1] + -31.210;
   1:  PR[91,2] = PR[90,2] + 12.457;
   1:  PR[91,3] = PR[90,3] + 15.535;
   1:L PR[91] R[100]mm/sec CNT100;
   1:  PR[91,1] = PR[90,1] + -31.797;
   1:  PR[91,2] = PR[90,2] + 11.847;
   1:  PR[91,3] = PR[90,3] + 15.540;
   1:L PR[91] R[100]mm/sec CNT100;
   1:  PR[91,1] = PR[90,1] + -32.352;
   1:  PR[91,2] = PR[90,2] + 11.209;
   1:  PR[91,3] = PR[90,3] + 15.546;
   1:L PR[91] R[100]mm/sec CNT100;
   1:  PR[91,1] = PR[90,1] + -32.877;
   1:  PR[91,2] = PR[90,2] + 10.541;
   1:  PR[91,3] = PR[90,3] + 15.551;
   1:L PR[91] R[100]mm/sec CNT100;
   1:  PR[91,1] = PR[90,1] + -33.360;
   1:  PR[91,2] = PR[90,2] + 9.858;
   1:  PR[91,3] = PR[90,3] + 15.557;
   1:L PR[91] R[100]mm/sec CNT100;
   1:  PR[91,1] = PR[90,1] + -33.812;
   1:  PR[91,2] = PR[90,2] + 9.147;
   1:  PR[91,3] = PR[90,3] + 15.563;
   1:L PR[91] R[100]mm/sec CNT100;
   1:  PR[91,1] = PR[90,1] + -34.228;
   1:  PR[91,2] = PR[90,2] + 8.415;
   1:  PR[91,3] = PR[90,3] + 15.568;
   1:L PR[91] R[100]mm/sec CNT100;
   1:  PR[91,1] = PR[90,1] + -34.607;
   1:  PR[91,2] = PR[90,2] + 7.667;
   1:  PR[91,3] = PR[90,3] + 15.574;
   1:L PR[91] R[100]mm/sec CNT100;
   1:  PR[91,1] = PR[90,1] + -34.948;
   1:  PR[91,2] = PR[90,2] + 6.904;
   1:  PR[91,3] = PR[90,3] + 15.579;
   1:L PR[91] R[100]mm/sec CNT100;
   1:  PR[91,1] = PR[90,1] + -35.251;
   1:  PR[91,2] = PR[90,2] + 6.131;
   1:  PR[91,3] = PR[90,3] + 15.585;
   1:L PR[91] R[100]mm/sec CNT100;
   1:  PR[91,1] = PR[90,1] + -35.514;
   1:  PR[91,2] = PR[90,2] + 5.349;
   1:  PR[91,3] = PR[90,3] + 15.591;
   1:L PR[91] R[100]mm/sec CNT100;
   1:  PR[91,1] = PR[90,1] + -35.738;
   1:  PR[91,2] = PR[90,2] + 4.559;
   1:  PR[91,3] = PR[90,3] + 15.596;
   1:L PR[91] R[100]mm/sec CNT100;
   1:  PR[91,1] = PR[90,1] + -35.921;
   1:  PR[91,2] = PR[90,2] + 3.760;
   1:  PR[91,3] = PR[90,3] + 15.601;
   1:L PR[91] R[100]mm/sec CNT100;
   1:  PR[91,1] = PR[90,1] + -36.064;
   1:  PR[91,2] = PR[90,2] + 2.950;
   1:  PR[91,3] = PR[90,3] + 15.607;
   1:L PR[91] R[100]mm/sec CNT100;
   1:  PR[91,1] = PR[90,1] + -36.167;
   1:  PR[91,2] = PR[90,2] + 2.126;
   1:  PR[91,3] = PR[90,3] + 15.612;
   1:L PR[91] R[100]mm/sec CNT100;
   1:  PR[91,1] = PR[90,1] + -36.229;
   1:  PR[91,2] = PR[90,2] + 1.286;
   1:  PR[91,3] = PR[90,3] + 15.618;
   1:L PR[91] R[100]mm/sec CNT100;
   1:  PR[91,1] = PR[90,1] + -36.249;
   1:  PR[91,2] = PR[90,2] + 0.428;
   1:  PR[91,3] = PR[90,3] + 15.624;
   1:L PR[91] R[100]mm/sec CNT100;
   1:  PR[91,1] = PR[90,1] + -36.229;
   1:  PR[91,2] = PR[90,2] + -0.431;
   1:  PR[91,3] = PR[90,3] + 15.629;
   1:L PR[91] R[100]mm/sec CNT100;
   1:  PR[91,1] = PR[90,1] + -36.167;
   1:  PR[91,2] = PR[90,2] + -1.271;
   1:  PR[91,3] = PR[90,3] + 15.635;
   1:L PR[91] R[100]mm/sec CNT100;
   1:  PR[91,1] = PR[90,1] + -36.064;
   1:  PR[91,2] = PR[90,2] + -2.095;
   1:  PR[91,3] = PR[90,3] + 15.641;
   1:L PR[91] R[100]mm/sec CNT100;
   1:  PR[91,1] = PR[90,1] + -35.921;
   1:  PR[91,2] = PR[90,2] + -2.905;
   1:  PR[91,3] = PR[90,3] + 15.646;
   1:L PR[91] R[100]mm/sec CNT100;
   1:  PR[91,1] = PR[90,1] + -35.738;
   1:  PR[91,2] = PR[90,2] + -3.704;
   1:  PR[91,3] = PR[90,3] + 15.652;
   1:L PR[91] R[100]mm/sec CNT100;
   1:  PR[91,1] = PR[90,1] + -35.514;
   1:  PR[91,2] = PR[90,2] + -4.494;
   1:  PR[91,3] = PR[90,3] + 15.657;
   1:L PR[91] R[100]mm/sec CNT100;
   1:  PR[91,1] = PR[90,1] + -35.251;
   1:  PR[91,2] = PR[90,2] + -5.276;
   1:  PR[91,3] = PR[90,3] + 15.663;
   1:L PR[91] R[100]mm/sec CNT100;
   1:  PR[91,1] = PR[90,1] + -34.948;
   1:  PR[91,2] = PR[90,2] + -6.049;
   1:  PR[91,3] = PR[90,3] + 15.668;
   1:L PR[91] R[100]mm/sec CNT100;
   1:  PR[91,1] = PR[90,1] + -34.607;
   1:  PR[91,2] = PR[90,2] + -6.811;
   1:  PR[91,3] = PR[90,3] + 15.674;
   1:L PR[91] R[100]mm/sec CNT100;
   1:  PR[91,1] = PR[90,1] + -34.228;
   1:  PR[91,2] = PR[90,2] + -7.560;
   1:  PR[91,3] = PR[90,3] + 15.679;
   1:L PR[91] R[100]mm/sec CNT100;
   1:  PR[91,1] = PR[90,1] + -33.812;
   1:  PR[91,2] = PR[90,2] + -8.291;
   1:  PR[91,3] = PR[90,3] + 15.685;
   1:L PR[91] R[100]mm/sec CNT100;
   1:  PR[91,1] = PR[90,1] + -33.360;
   1:  PR[91,2] = PR[90,2] + -9.002;
   1:  PR[91,3] = PR[90,3] + 15.690;
   1:L PR[91] R[100]mm/sec CNT100;
   1:  PR[91,1] = PR[90,1] + -32.874;
   1:  PR[91,2] = PR[90,2] + -9.691;
   1:  PR[91,3] = PR[90,3] + 15.696;
   1:L PR[91] R[100]mm/sec CNT100;
   1:  PR[91,1] = PR[90,1] + -32.352;
   1:  PR[91,2] = PR[90,2] + -10.354;
   1:  PR[91,3] = PR[90,3] + 15.701;
   1:L PR[91] R[100]mm/sec CNT100;
   1:  PR[91,1] = PR[90,1] + -31.797;
   1:  PR[91,2] = PR[90,2] + -10.992;
   1:  PR[91,3] = PR[90,3] + 15.707;
   1:L PR[91] R[100]mm/sec CNT100;
   1:  PR[91,1] = PR[90,1] + -31.210;
   1:  PR[91,2] = PR[90,2] + -11.602;
   1:  PR[91,3] = PR[90,3] + 15.713;
   1:L PR[91] R[100]mm/sec CNT100;
   1:  PR[91,1] = PR[90,1] + -30.593;
   1:  PR[91,2] = PR[90,2] + -12.184;
   1:  PR[91,3] = PR[90,3] + 15.718;
   1:L PR[91] R[100]mm/sec CNT100;
   1:  PR[91,1] = PR[90,1] + -29.946;
   1:  PR[91,2] = PR[90,2] + -12.736;
   1:  PR[91,3] = PR[90,3] + 15.724;
   1:L PR[91] R[100]mm/sec CNT100;
   1:  PR[91,1] = PR[90,1] + -29.271;
   1:  PR[91,2] = PR[90,2] + -13.257;
   1:  PR[91,3] = PR[90,3] + 15.730;
   1:L PR[91] R[100]mm/sec CNT100;
   1:  PR[91,1] = PR[90,1] + -28.569;
   1:  PR[91,2] = PR[90,2] + -13.747;
   1:  PR[91,3] = PR[90,3] + 15.735;
   1:L PR[91] R[100]mm/sec CNT100;
   1:  PR[91,1] = PR[90,1] + -28.202;
   1:  PR[91,2] = PR[90,2] + -13.978;
   1:  PR[91,3] = PR[90,3] + 15.741;
   1:L PR[91] R[100]mm/sec CNT100;
   1:  PR[91,1] = PR[90,1] + -27.844;
   1:  PR[91,2] = PR[90,2] + -14.202;
   1:  PR[91,3] = PR[90,3] + 15.744;
   1:L PR[91] R[100]mm/sec CNT100;
   1:  PR[91,1] = PR[90,1] + -27.093;
   1:  PR[91,2] = PR[90,2] + -14.623;
   1:  PR[91,3] = PR[90,3] + 15.747;
   1:L PR[91] R[100]mm/sec CNT100;
   1:  PR[91,1] = PR[90,1] + -26.321;
   1:  PR[91,2] = PR[90,2] + -15.009;
   1:  PR[91,3] = PR[90,3] + 15.752;
   1:L PR[91] R[100]mm/sec CNT100;
   1:  PR[91,1] = PR[90,1] + -25.530;
   1:  PR[91,2] = PR[90,2] + -15.358;
   1:  PR[91,3] = PR[90,3] + 15.758;
   1:L PR[91] R[100]mm/sec CNT100;
   1:  PR[91,1] = PR[90,1] + -24.721;
   1:  PR[91,2] = PR[90,2] + -15.669;
   1:  PR[91,3] = PR[90,3] + 15.764;
   1:L PR[91] R[100]mm/sec CNT100;
   1:  PR[91,1] = PR[90,1] + -23.893;
   1:  PR[91,2] = PR[90,2] + -15.941;
   1:  PR[91,3] = PR[90,3] + 15.770;
   1:L PR[91] R[100]mm/sec CNT100;
   1:  PR[91,1] = PR[90,1] + -23.051;
   1:  PR[91,2] = PR[90,2] + -16.173;
   1:  PR[91,3] = PR[90,3] + 15.776;
   1:L PR[91] R[100]mm/sec CNT100;
   1:  PR[91,1] = PR[90,1] + -22.194;
   1:  PR[91,2] = PR[90,2] + -16.364;
   1:  PR[91,3] = PR[90,3] + 15.781;
   1:L PR[91] R[100]mm/sec CNT100;
   1:  PR[91,1] = PR[90,1] + -21.326;
   1:  PR[91,2] = PR[90,2] + -16.515;
   1:  PR[91,3] = PR[90,3] + 15.787;
   1:L PR[91] R[100]mm/sec CNT100;
   1:  PR[91,1] = PR[90,1] + -20.448;
   1:  PR[91,2] = PR[90,2] + -16.623;
   1:  PR[91,3] = PR[90,3] + 15.793;
   1:L PR[91] R[100]mm/sec CNT100;
   1:  PR[91,1] = PR[90,1] + -20.011;
   1:  PR[91,2] = PR[90,2] + -16.658;
   1:  PR[91,3] = PR[90,3] + 15.799;
   1:L PR[91] R[100]mm/sec CNT100;
   1:  PR[91,1] = PR[90,1] + -19.567;
   1:  PR[91,2] = PR[90,2] + -16.689;
   1:  PR[91,3] = PR[90,3] + 15.802;
   1:L PR[91] R[100]mm/sec CNT100;
   1:  PR[91,1] = PR[90,1] + -18.679;
   1:  PR[91,2] = PR[90,2] + -16.712;
   1:  PR[91,3] = PR[90,3] + 15.805;
   1:L PR[91] R[100]mm/sec CNT100;
   1:  PR[91,1] = PR[90,1] + -17.789;
   1:  PR[91,2] = PR[90,2] + -16.692;
   1:  PR[91,3] = PR[90,3] + 15.811;
   1:L PR[91] R[100]mm/sec CNT100;
   1:  PR[91,1] = PR[90,1] + -16.899;
   1:  PR[91,2] = PR[90,2] + -16.628;
   1:  PR[91,3] = PR[90,3] + 15.817;
   1:L PR[91] R[100]mm/sec CNT100;
   1:  PR[91,1] = PR[90,1] + -16.052;
   1:  PR[91,2] = PR[90,2] + -16.527;
   1:  PR[91,3] = PR[90,3] + 15.823;
   1:L PR[91] R[100]mm/sec CNT100;
   1:  PR[91,1] = PR[90,1] + -15.240;
   1:  PR[91,2] = PR[90,2] + -16.393;
   1:  PR[91,3] = PR[90,3] + 15.828;
   1:L PR[91] R[100]mm/sec CNT100;
   1:  PR[91,1] = PR[90,1] + -14.125;
   1:  PR[91,2] = PR[90,2] + -16.147;
   1:  PR[91,3] = PR[90,3] + 15.834;
   1:L PR[91] R[100]mm/sec CNT100;
   1:  PR[91,1] = PR[90,1] + -13.222;
   1:  PR[91,2] = PR[90,2] + -15.894;
   1:  PR[91,3] = PR[90,3] + 15.841;
   1:L PR[91] R[100]mm/sec CNT100;
   1:  PR[91,1] = PR[90,1] + -12.335;
   1:  PR[91,2] = PR[90,2] + -15.595;
   1:  PR[91,3] = PR[90,3] + 15.848;
   1:L PR[91] R[100]mm/sec CNT100;
   1:  PR[91,1] = PR[90,1] + -11.342;
   1:  PR[91,2] = PR[90,2] + -15.199;
   1:  PR[91,3] = PR[90,3] + 15.854;
   1:L PR[91] R[100]mm/sec CNT100;
   1:  PR[91,1] = PR[90,1] + -10.612;
   1:  PR[91,2] = PR[90,2] + -14.864;
   1:  PR[91,3] = PR[90,3] + 15.861;
   1:L PR[91] R[100]mm/sec CNT100;
   1:  PR[91,1] = PR[90,1] + -9.820;
   1:  PR[91,2] = PR[90,2] + -14.456;
   1:  PR[91,3] = PR[90,3] + 15.866;
   1:L PR[91] R[100]mm/sec CNT100;
   1:  PR[91,1] = PR[90,1] + -9.043;
   1:  PR[91,2] = PR[90,2] + -14.008;
   1:  PR[91,3] = PR[90,3] + 15.872;
   1:L PR[91] R[100]mm/sec CNT100;
   1:  PR[91,1] = PR[90,1] + -8.290;
   1:  PR[91,2] = PR[90,2] + -13.522;
   1:  PR[91,3] = PR[90,3] + 15.878;
   1:L PR[91] R[100]mm/sec CNT100;
   1:  PR[91,1] = PR[90,1] + -7.561;
   1:  PR[91,2] = PR[90,2] + -12.998;
   1:  PR[91,3] = PR[90,3] + 15.884;
   1:L PR[91] R[100]mm/sec CNT100;
   1:  PR[91,1] = PR[90,1] + -7.302;
   1:  PR[91,2] = PR[90,2] + -12.795;
   1:  PR[91,3] = PR[90,3] + 15.890;
   1:L PR[91] R[100]mm/sec CNT100;
   1:  PR[91,1] = PR[90,1] + -6.863;
   1:  PR[91,2] = PR[90,2] + -12.443;
   1:  PR[91,3] = PR[90,3] + 15.892;
   1:L PR[91] R[100]mm/sec CNT100;
   1:  PR[91,1] = PR[90,1] + -6.192;
   1:  PR[91,2] = PR[90,2] + -11.850;
   1:  PR[91,3] = PR[90,3] + 15.896;
   1:L PR[91] R[100]mm/sec CNT100;
   1:  PR[91,1] = PR[90,1] + -5.548;
   1:  PR[91,2] = PR[90,2] + -11.219;
   1:  PR[91,3] = PR[90,3] + 15.902;
   1:L PR[91] R[100]mm/sec CNT100;
   1:  PR[91,1] = PR[90,1] + -4.945;
   1:  PR[91,2] = PR[90,2] + -10.566;
   1:  PR[91,3] = PR[90,3] + 15.908;
   1:L PR[91] R[100]mm/sec CNT100;
   1:  PR[91,1] = PR[90,1] + -4.371;
   1:  PR[91,2] = PR[90,2] + -9.876;
   1:  PR[91,3] = PR[90,3] + 15.914;
   1:L PR[91] R[100]mm/sec CNT100;
   1:  PR[91,1] = PR[90,1] + -4.015;
   1:  PR[91,2] = PR[90,2] + -9.402;
   1:  PR[91,3] = PR[90,3] + 15.920;
   1:L PR[91] R[100]mm/sec CNT100;
   1:  PR[91,1] = PR[90,1] + -3.339;
   1:  PR[91,2] = PR[90,2] + -8.410;
   1:  PR[91,3] = PR[90,3] + 15.924;
   1:L PR[91] R[100]mm/sec CNT100;
   1:  PR[91,1] = PR[90,1] + -2.505;
   1:  PR[91,2] = PR[90,2] + -6.986;
   1:  PR[91,3] = PR[90,3] + 15.932;
   1:L PR[91] R[100]mm/sec CNT100;
   1:  PR[91,1] = PR[90,1] + -2.231;
   1:  PR[91,2] = PR[90,2] + -6.641;
   1:  PR[91,3] = PR[90,3] + 15.943;
   1:L PR[91] R[100]mm/sec CNT100;
   1:  PR[91,1] = PR[90,1] + -1.914;
   1:  PR[91,2] = PR[90,2] + -6.332;
   1:  PR[91,3] = PR[90,3] + 15.946;
   1:L PR[91] R[100]mm/sec CNT100;
   1:  PR[91,1] = PR[90,1] + -1.543;
   1:  PR[91,2] = PR[90,2] + -6.062;
   1:  PR[91,3] = PR[90,3] + 15.949;
   1:L PR[91] R[100]mm/sec CNT100;
   1:  PR[91,1] = PR[90,1] + -1.206;
   1:  PR[91,2] = PR[90,2] + -5.882;
   1:  PR[91,3] = PR[90,3] + 15.952;
   1:L PR[91] R[100]mm/sec CNT100;
   1:  PR[91,1] = PR[90,1] + -0.808;
   1:  PR[91,2] = PR[90,2] + -5.739;
   1:  PR[91,3] = PR[90,3] + 15.954;
   1:L PR[91] R[100]mm/sec CNT100;
   1:  PR[91,1] = PR[90,1] + -0.384;
   1:  PR[91,2] = PR[90,2] + -5.660;
   1:  PR[91,3] = PR[90,3] + 15.957;
   1:L PR[91] R[100]mm/sec CNT100;
   1:  PR[91] = PR[90];
   1:  PR[91,1] = PR[90,1] + 0.086;
   1:  PR[91,2] = PR[90,2] + -6.637;
   1:  PR[91,3] = PR[90,3] + 17.290;
   1:L PR[91] R[100]mm/sec CNT100;
   1:  PR[91,1] = PR[90,1] + 0.493;
   1:  PR[91,2] = PR[90,2] + -6.701;
   1:  PR[91,3] = PR[90,3] + 15.963;
   1:L PR[91] R[100]mm/sec CNT100;
   1:  PR[91,1] = PR[90,1] + 0.889;
   1:  PR[91,2] = PR[90,2] + -6.828;
   1:  PR[91,3] = PR[90,3] + 15.966;
   1:L PR[91] R[100]mm/sec CNT100;
   1:  PR[91,1] = PR[90,1] + 1.270;
   1:  PR[91,2] = PR[90,2] + -7.017;
   1:  PR[91,3] = PR[90,3] + 15.968;
   1:L PR[91] R[100]mm/sec CNT100;
   1:  PR[91,1] = PR[90,1] + 1.583;
   1:  PR[91,2] = PR[90,2] + -7.229;
   1:  PR[91,3] = PR[90,3] + 15.971;
   1:L PR[91] R[100]mm/sec CNT100;
   1:  PR[91,1] = PR[90,1] + 1.895;
   1:  PR[91,2] = PR[90,2] + -7.504;
   1:  PR[91,3] = PR[90,3] + 15.974;
   1:L PR[91] R[100]mm/sec CNT100;
   1:  PR[91,1] = PR[90,1] + 2.254;
   1:  PR[91,2] = PR[90,2] + -7.933;
   1:  PR[91,3] = PR[90,3] + 15.977;
   1:L PR[91] R[100]mm/sec CNT100;
   1:  PR[91,1] = PR[90,1] + 2.853;
   1:  PR[91,2] = PR[90,2] + -8.863;
   1:  PR[91,3] = PR[90,3] + 15.980;
   1:L PR[91] R[100]mm/sec CNT100;
   1:  PR[91,1] = PR[90,1] + 3.286;
   1:  PR[91,2] = PR[90,2] + -9.474;
   1:  PR[91,3] = PR[90,3] + 15.988;
   1:L PR[91] R[100]mm/sec CNT100;
   1:  PR[91,1] = PR[90,1] + 3.946;
   1:  PR[91,2] = PR[90,2] + -10.314;
   1:  PR[91,3] = PR[90,3] + 15.993;
   1:L PR[91] R[100]mm/sec CNT100;
   1:  PR[91,1] = PR[90,1] + 4.555;
   1:  PR[91,2] = PR[90,2] + -11.002;
   1:  PR[91,3] = PR[90,3] + 16.000;
   1:L PR[91] R[100]mm/sec CNT100;
   1:  PR[91,1] = PR[90,1] + 4.838;
   1:  PR[91,2] = PR[90,2] + -11.296;
   1:  PR[91,3] = PR[90,3] + 16.006;
   1:L PR[91] R[100]mm/sec CNT100;
   1:  PR[91,1] = PR[90,1] + 5.199;
   1:  PR[91,2] = PR[90,2] + -11.655;
   1:  PR[91,3] = PR[90,3] + 16.009;
   1:L PR[91] R[100]mm/sec CNT100;
   1:  PR[91,1] = PR[90,1] + 5.887;
   1:  PR[91,2] = PR[90,2] + -12.283;
   1:  PR[91,3] = PR[90,3] + 16.013;
   1:L PR[91] R[100]mm/sec CNT100;
   1:  PR[91,1] = PR[90,1] + 6.636;
   1:  PR[91,2] = PR[90,2] + -12.894;
   1:  PR[91,3] = PR[90,3] + 16.019;
   1:L PR[91] R[100]mm/sec CNT100;
   1:  PR[91,1] = PR[90,1] + 7.354;
   1:  PR[91,2] = PR[90,2] + -13.422;
   1:  PR[91,3] = PR[90,3] + 16.025;
   1:L PR[91] R[100]mm/sec CNT100;
   1:  PR[91,1] = PR[90,1] + 7.920;
   1:  PR[91,2] = PR[90,2] + -13.799;
   1:  PR[91,3] = PR[90,3] + 16.031;
   1:L PR[91] R[100]mm/sec CNT100;
   1:  PR[91,1] = PR[90,1] + 8.906;
   1:  PR[91,2] = PR[90,2] + -14.394;
   1:  PR[91,3] = PR[90,3] + 16.036;
   1:L PR[91] R[100]mm/sec CNT100;
   1:  PR[91,1] = PR[90,1] + 9.712;
   1:  PR[91,2] = PR[90,2] + -14.818;
   1:  PR[91,3] = PR[90,3] + 16.044;
   1:L PR[91] R[100]mm/sec CNT100;
   1:  PR[91,1] = PR[90,1] + 10.694;
   1:  PR[91,2] = PR[90,2] + -15.267;
   1:  PR[91,3] = PR[90,3] + 16.050;
   1:L PR[91] R[100]mm/sec CNT100;
   1:  PR[91,1] = PR[90,1] + 11.392;
   1:  PR[91,2] = PR[90,2] + -15.550;
   1:  PR[91,3] = PR[90,3] + 16.057;
   1:L PR[91] R[100]mm/sec CNT100;
   1:  PR[91,1] = PR[90,1] + 12.250;
   1:  PR[91,2] = PR[90,2] + -15.853;
   1:  PR[91,3] = PR[90,3] + 16.062;
   1:L PR[91] R[100]mm/sec CNT100;
   1:  PR[91,1] = PR[90,1] + 13.120;
   1:  PR[91,2] = PR[90,2] + -16.113;
   1:  PR[91,3] = PR[90,3] + 16.068;
   1:L PR[91] R[100]mm/sec CNT100;
   1:  PR[91,1] = PR[90,1] + 13.660;
   1:  PR[91,2] = PR[90,2] + -16.249;
   1:  PR[91,3] = PR[90,3] + 16.075;
   1:L PR[91] R[100]mm/sec CNT100;
   1:  PR[91,1] = PR[90,1] + 13.996;
   1:  PR[91,2] = PR[90,2] + -16.330;
   1:  PR[91,3] = PR[90,3] + 16.078;
   1:L PR[91] R[100]mm/sec CNT100;
   1:  PR[91,1] = PR[90,1] + 14.881;
   1:  PR[91,2] = PR[90,2] + -16.504;
   1:  PR[91,3] = PR[90,3] + 16.081;
   1:L PR[91] R[100]mm/sec CNT100;
   1:  PR[91,1] = PR[90,1] + 15.964;
   1:  PR[91,2] = PR[90,2] + -16.656;
   1:  PR[91,3] = PR[90,3] + 16.087;
   1:L PR[91] R[100]mm/sec CNT100;
   1:  PR[91,1] = PR[90,1] + 16.669;
   1:  PR[91,2] = PR[90,2] + -16.723;
   1:  PR[91,3] = PR[90,3] + 16.094;
   1:L PR[91] R[100]mm/sec CNT100;
   1:  PR[91,1] = PR[90,1] + 17.536;
   1:  PR[91,2] = PR[90,2] + -16.767;
   1:  PR[91,3] = PR[90,3] + 16.099;
   1:L PR[91] R[100]mm/sec CNT100;
   1:  PR[91,1] = PR[90,1] + 18.358;
   1:  PR[91,2] = PR[90,2] + -16.771;
   1:  PR[91,3] = PR[90,3] + 16.105;
   1:L PR[91] R[100]mm/sec CNT100;
   1:  PR[91,1] = PR[90,1] + 19.184;
   1:  PR[91,2] = PR[90,2] + -16.738;
   1:  PR[91,3] = PR[90,3] + 16.110;
   1:L PR[91] R[100]mm/sec CNT100;
   1:  PR[91,1] = PR[90,1] + 20.011;
   1:  PR[91,2] = PR[90,2] + -16.669;
   1:  PR[91,3] = PR[90,3] + 16.116;
   1:L PR[91] R[100]mm/sec CNT100;
   1:  PR[91,1] = PR[90,1] + 20.836;
   1:  PR[91,2] = PR[90,2] + -16.562;
   1:  PR[91,3] = PR[90,3] + 16.122;
   1:L PR[91] R[100]mm/sec CNT100;
   1:  PR[91,1] = PR[90,1] + 21.658;
   1:  PR[91,2] = PR[90,2] + -16.418;
   1:  PR[91,3] = PR[90,3] + 16.127;
   1:L PR[91] R[100]mm/sec CNT100;
   1:  PR[91,1] = PR[90,1] + 22.476;
   1:  PR[91,2] = PR[90,2] + -16.235;
   1:  PR[91,3] = PR[90,3] + 16.133;
   1:L PR[91] R[100]mm/sec CNT100;
   1:  PR[91,1] = PR[90,1] + 23.287;
   1:  PR[91,2] = PR[90,2] + -16.015;
   1:  PR[91,3] = PR[90,3] + 16.138;
   1:L PR[91] R[100]mm/sec CNT100;
   1:  PR[91,1] = PR[90,1] + 24.097;
   1:  PR[91,2] = PR[90,2] + -15.754;
   1:  PR[91,3] = PR[90,3] + 16.144;
   1:L PR[91] R[100]mm/sec CNT100;
   1:  PR[91,1] = PR[90,1] + 24.921;
   1:  PR[91,2] = PR[90,2] + -15.444;
   1:  PR[91,3] = PR[90,3] + 16.150;
   1:L PR[91] R[100]mm/sec CNT100;
   1:  PR[91,1] = PR[90,1] + 25.727;
   1:  PR[91,2] = PR[90,2] + -15.096;
   1:  PR[91,3] = PR[90,3] + 16.156;
   1:L PR[91] R[100]mm/sec CNT100;
   1:  PR[91,1] = PR[90,1] + 26.512;
   1:  PR[91,2] = PR[90,2] + -14.710;
   1:  PR[91,3] = PR[90,3] + 16.162;
   1:L PR[91] R[100]mm/sec CNT100;
   1:  PR[91,1] = PR[90,1] + 27.275;
   1:  PR[91,2] = PR[90,2] + -14.289;
   1:  PR[91,3] = PR[90,3] + 16.168;
   1:L PR[91] R[100]mm/sec CNT100;
   1:  PR[91,1] = PR[90,1] + 28.013;
   1:  PR[91,2] = PR[90,2] + -13.832;
   1:  PR[91,3] = PR[90,3] + 16.174;
   1:L PR[91] R[100]mm/sec CNT100;
   1:  PR[91,1] = PR[90,1] + 28.726;
   1:  PR[91,2] = PR[90,2] + -13.341;
   1:  PR[91,3] = PR[90,3] + 16.179;
   1:L PR[91] R[100]mm/sec CNT100;
   1:  PR[91,1] = PR[90,1] + 29.412;
   1:  PR[91,2] = PR[90,2] + -12.817;
   1:  PR[91,3] = PR[90,3] + 16.185;
   1:L PR[91] R[100]mm/sec CNT100;
   1:  PR[91,1] = PR[90,1] + 30.070;
   1:  PR[91,2] = PR[90,2] + -12.262;
   1:  PR[91,3] = PR[90,3] + 16.191;
   1:L PR[91] R[100]mm/sec CNT100;
   1:  PR[91,1] = PR[90,1] + 30.697;
   1:  PR[91,2] = PR[90,2] + -11.677;
   1:  PR[91,3] = PR[90,3] + 16.197;
   1:L PR[91] R[100]mm/sec CNT100;
   1:  PR[91,1] = PR[90,1] + 31.293;
   1:  PR[91,2] = PR[90,2] + -11.061;
   1:  PR[91,3] = PR[90,3] + 16.203;
   1:L PR[91] R[100]mm/sec CNT100;
   1:  PR[91,1] = PR[90,1] + 31.868;
   1:  PR[91,2] = PR[90,2] + -10.404;
   1:  PR[91,3] = PR[90,3] + 16.209;
   1:L PR[91] R[100]mm/sec CNT100;
   1:  PR[91,1] = PR[90,1] + 32.386;
   1:  PR[91,2] = PR[90,2] + -9.749;
   1:  PR[91,3] = PR[90,3] + 16.214;
   1:L PR[91] R[100]mm/sec CNT100;
   1:  PR[91,1] = PR[90,1] + 32.879;
   1:  PR[91,2] = PR[90,2] + -9.055;
   1:  PR[91,3] = PR[90,3] + 16.220;
   1:L PR[91] R[100]mm/sec CNT100;
   1:  PR[91,1] = PR[90,1] + 33.338;
   1:  PR[91,2] = PR[90,2] + -8.339;
   1:  PR[91,3] = PR[90,3] + 16.226;
   1:L PR[91] R[100]mm/sec CNT100;
   1:  PR[91,1] = PR[90,1] + 33.760;
   1:  PR[91,2] = PR[90,2] + -7.604;
   1:  PR[91,3] = PR[90,3] + 16.232;
   1:L PR[91] R[100]mm/sec CNT100;
   1:  PR[91,1] = PR[90,1] + 34.144;
   1:  PR[91,2] = PR[90,2] + -6.853;
   1:  PR[91,3] = PR[90,3] + 16.237;
   1:L PR[91] R[100]mm/sec CNT100;
   1:  PR[91,1] = PR[90,1] + 34.491;
   1:  PR[91,2] = PR[90,2] + -6.090;
   1:  PR[91,3] = PR[90,3] + 16.243;
   1:L PR[91] R[100]mm/sec CNT100;
   1:  PR[91,1] = PR[90,1] + 34.798;
   1:  PR[91,2] = PR[90,2] + -5.317;
   1:  PR[91,3] = PR[90,3] + 16.249;
   1:L PR[91] R[100]mm/sec CNT100;
   1:  PR[91,1] = PR[90,1] + 35.065;
   1:  PR[91,2] = PR[90,2] + -4.535;
   1:  PR[91,3] = PR[90,3] + 16.254;
   1:L PR[91] R[100]mm/sec CNT100;
   1:  PR[91,1] = PR[90,1] + 35.291;
   1:  PR[91,2] = PR[90,2] + -3.742;
   1:  PR[91,3] = PR[90,3] + 16.260;
   1:L PR[91] R[100]mm/sec CNT100;
   1:  PR[91,1] = PR[90,1] + 35.477;
   1:  PR[91,2] = PR[90,2] + -2.940;
   1:  PR[91,3] = PR[90,3] + 16.265;
   1:L PR[91] R[100]mm/sec CNT100;
   1:  PR[91,1] = PR[90,1] + 35.623;
   1:  PR[91,2] = PR[90,2] + -2.123;
   1:  PR[91,3] = PR[90,3] + 16.271;
   1:L PR[91] R[100]mm/sec CNT100;
   1:  PR[91,1] = PR[90,1] + 35.727;
   1:  PR[91,2] = PR[90,2] + -1.292;
   1:  PR[91,3] = PR[90,3] + 16.277;
   1:L PR[91] R[100]mm/sec CNT100;
   1:  PR[91,1] = PR[90,1] + 35.789;
   1:  PR[91,2] = PR[90,2] + -0.441;
   1:  PR[91,3] = PR[90,3] + 16.282;
   1:L PR[91] R[100]mm/sec CNT100;
   1:  PR[91,1] = PR[90,1] + 35.812;
   1:  PR[91,2] = PR[90,2] + 0.428;
   1:  PR[91,3] = PR[90,3] + 16.288;
   1:L PR[91] R[100]mm/sec CNT100;
   1:  PR[91,1] = PR[90,1] + 35.789;
   1:  PR[91,2] = PR[90,2] + 1.296;
   1:  PR[91,3] = PR[90,3] + 16.294;
   1:L PR[91] R[100]mm/sec CNT100;
   1:  PR[91,1] = PR[90,1] + 35.727;
   1:  PR[91,2] = PR[90,2] + 2.147;
   1:  PR[91,3] = PR[90,3] + 16.300;
   1:L PR[91] R[100]mm/sec CNT100;
   1:  PR[91,1] = PR[90,1] + 35.623;
   1:  PR[91,2] = PR[90,2] + 2.979;
   1:  PR[91,3] = PR[90,3] + 16.306;
   1:L PR[91] R[100]mm/sec CNT100;
   1:  PR[91,1] = PR[90,1] + 35.477;
   1:  PR[91,2] = PR[90,2] + 3.795;
   1:  PR[91,3] = PR[90,3] + 16.311;
   1:L PR[91] R[100]mm/sec CNT100;
   1:  PR[91,1] = PR[90,1] + 35.291;
   1:  PR[91,2] = PR[90,2] + 4.598;
   1:  PR[91,3] = PR[90,3] + 16.317;
   1:L PR[91] R[100]mm/sec CNT100;
   1:  PR[91,1] = PR[90,1] + 35.065;
   1:  PR[91,2] = PR[90,2] + 5.390;
   1:  PR[91,3] = PR[90,3] + 16.322;
   1:L PR[91] R[100]mm/sec CNT100;
   1:  PR[91,1] = PR[90,1] + 34.798;
   1:  PR[91,2] = PR[90,2] + 6.172;
   1:  PR[91,3] = PR[90,3] + 16.328;
   1:L PR[91] R[100]mm/sec CNT100;
   1:  PR[91,1] = PR[90,1] + 34.491;
   1:  PR[91,2] = PR[90,2] + 6.945;
   1:  PR[91,3] = PR[90,3] + 16.334;
   1:L PR[91] R[100]mm/sec CNT100;
   1:  PR[91,1] = PR[90,1] + 34.145;
   1:  PR[91,2] = PR[90,2] + 7.708;
   1:  PR[91,3] = PR[90,3] + 16.339;
   1:L PR[91] R[100]mm/sec CNT100;
   1:  PR[91,1] = PR[90,1] + 33.760;
   1:  PR[91,2] = PR[90,2] + 8.459;
   1:  PR[91,3] = PR[90,3] + 16.345;
   1:L PR[91] R[100]mm/sec CNT100;
   1:  PR[91,1] = PR[90,1] + 33.338;
   1:  PR[91,2] = PR[90,2] + 9.194;
   1:  PR[91,3] = PR[90,3] + 16.351;
   1:L PR[91] R[100]mm/sec CNT100;
   1:  PR[91,1] = PR[90,1] + 32.879;
   1:  PR[91,2] = PR[90,2] + 9.910;
   1:  PR[91,3] = PR[90,3] + 16.356;
   1:L PR[91] R[100]mm/sec CNT100;
   1:  PR[91,1] = PR[90,1] + 32.386;
   1:  PR[91,2] = PR[90,2] + 10.604;
   1:  PR[91,3] = PR[90,3] + 16.362;
   1:L PR[91] R[100]mm/sec CNT100;
   1:  PR[91,1] = PR[90,1] + 31.857;
   1:  PR[91,2] = PR[90,2] + 11.273;
   1:  PR[91,3] = PR[90,3] + 16.368;
   1:L PR[91] R[100]mm/sec CNT100;
   1:  PR[91,1] = PR[90,1] + 31.293;
   1:  PR[91,2] = PR[90,2] + 11.916;
   1:  PR[91,3] = PR[90,3] + 16.373;
   1:L PR[91] R[100]mm/sec CNT100;
   1:  PR[91,1] = PR[90,1] + 30.697;
   1:  PR[91,2] = PR[90,2] + 12.532;
   1:  PR[91,3] = PR[90,3] + 16.379;
   1:L PR[91] R[100]mm/sec CNT100;
   1:  PR[91,1] = PR[90,1] + 30.070;
   1:  PR[91,2] = PR[90,2] + 13.118;
   1:  PR[91,3] = PR[90,3] + 16.385;
   1:L PR[91] R[100]mm/sec CNT100;
   1:  PR[91,1] = PR[90,1] + 29.412;
   1:  PR[91,2] = PR[90,2] + 13.673;
   1:  PR[91,3] = PR[90,3] + 16.391;
   1:L PR[91] R[100]mm/sec CNT100;
   1:  PR[91,1] = PR[90,1] + 28.726;
   1:  PR[91,2] = PR[90,2] + 14.197;
   1:  PR[91,3] = PR[90,3] + 16.397;
   1:L PR[91] R[100]mm/sec CNT100;
   1:  PR[91,1] = PR[90,1] + 28.321;
   1:  PR[91,2] = PR[90,2] + 14.477;
   1:  PR[91,3] = PR[90,3] + 16.403;
   1:L PR[91] R[100]mm/sec CNT100;
   1:  PR[91,1] = PR[90,1] + 28.014;
   1:  PR[91,2] = PR[90,2] + 14.686;
   1:  PR[91,3] = PR[90,3] + 16.406;
   1:L PR[91] R[100]mm/sec CNT100;
   1:  PR[91,1] = PR[90,1] + 27.277;
   1:  PR[91,2] = PR[90,2] + 15.142;
   1:  PR[91,3] = PR[90,3] + 16.408;
   1:L PR[91] R[100]mm/sec CNT100;
   1:  PR[91,1] = PR[90,1] + 26.263;
   1:  PR[91,2] = PR[90,2] + 15.688;
   1:  PR[91,3] = PR[90,3] + 16.414;
   1:L PR[91] R[100]mm/sec CNT100;
   1:  PR[91,1] = PR[90,1] + 25.727;
   1:  PR[91,2] = PR[90,2] + 15.951;
   1:  PR[91,3] = PR[90,3] + 16.422;
   1:L PR[91] R[100]mm/sec CNT100;
   1:  PR[91,1] = PR[90,1] + 24.921;
   1:  PR[91,2] = PR[90,2] + 16.299;
   1:  PR[91,3] = PR[90,3] + 16.426;
   1:L PR[91] R[100]mm/sec CNT100;
   1:  PR[91,1] = PR[90,1] + 24.077;
   1:  PR[91,2] = PR[90,2] + 16.615;
   1:  PR[91,3] = PR[90,3] + 16.432;
   1:L PR[91] R[100]mm/sec CNT100;
   1:  PR[91,1] = PR[90,1] + 23.287;
   1:  PR[91,2] = PR[90,2] + 16.870;
   1:  PR[91,3] = PR[90,3] + 16.438;
   1:L PR[91] R[100]mm/sec CNT100;
   1:  PR[91,1] = PR[90,1] + 22.476;
   1:  PR[91,2] = PR[90,2] + 17.090;
   1:  PR[91,3] = PR[90,3] + 16.444;
   1:L PR[91] R[100]mm/sec CNT100;
   1:  PR[91,1] = PR[90,1] + 21.658;
   1:  PR[91,2] = PR[90,2] + 17.273;
   1:  PR[91,3] = PR[90,3] + 16.449;
   1:L PR[91] R[100]mm/sec CNT100;
   1:  PR[91,1] = PR[90,1] + 20.836;
   1:  PR[91,2] = PR[90,2] + 17.417;
   1:  PR[91,3] = PR[90,3] + 16.455;
   1:L PR[91] R[100]mm/sec CNT100;
   1:  PR[91,1] = PR[90,1] + 20.009;
   1:  PR[91,2] = PR[90,2] + 17.524;
   1:  PR[91,3] = PR[90,3] + 16.461;
   1:L PR[91] R[100]mm/sec CNT100;
   1:  PR[91,1] = PR[90,1] + 19.488;
   1:  PR[91,2] = PR[90,2] + 17.572;
   1:  PR[91,3] = PR[90,3] + 16.466;
   1:L PR[91] R[100]mm/sec CNT100;
   1:  PR[91,1] = PR[90,1] + 18.356;
   1:  PR[91,2] = PR[90,2] + 17.626;
   1:  PR[91,3] = PR[90,3] + 16.470;
   1:L PR[91] R[100]mm/sec CNT100;
   1:  PR[91,1] = PR[90,1] + 17.536;
   1:  PR[91,2] = PR[90,2] + 17.622;
   1:  PR[91,3] = PR[90,3] + 16.477;
   1:L PR[91] R[100]mm/sec CNT100;
   1:  PR[91,1] = PR[90,1] + 16.670;
   1:  PR[91,2] = PR[90,2] + 17.578;
   1:  PR[91,3] = PR[90,3] + 16.483;
   1:L PR[91] R[100]mm/sec CNT100;
   1:  PR[91,1] = PR[90,1] + 15.775;
   1:  PR[91,2] = PR[90,2] + 17.491;
   1:  PR[91,3] = PR[90,3] + 16.489;
   1:L PR[91] R[100]mm/sec CNT100;
   1:  PR[91,1] = PR[90,1] + 14.883;
   1:  PR[91,2] = PR[90,2] + 17.360;
   1:  PR[91,3] = PR[90,3] + 16.495;
   1:L PR[91] R[100]mm/sec CNT100;
   1:  PR[91,1] = PR[90,1] + 13.996;
   1:  PR[91,2] = PR[90,2] + 17.185;
   1:  PR[91,3] = PR[90,3] + 16.501;
   1:L PR[91] R[100]mm/sec CNT100;
   1:  PR[91,1] = PR[90,1] + 13.659;
   1:  PR[91,2] = PR[90,2] + 17.104;
   1:  PR[91,3] = PR[90,3] + 16.507;
   1:L PR[91] R[100]mm/sec CNT100;
   1:  PR[91,1] = PR[90,1] + 13.120;
   1:  PR[91,2] = PR[90,2] + 16.968;
   1:  PR[91,3] = PR[90,3] + 16.509;
   1:L PR[91] R[100]mm/sec CNT100;
   1:  PR[91,1] = PR[90,1] + 12.250;
   1:  PR[91,2] = PR[90,2] + 16.708;
   1:  PR[91,3] = PR[90,3] + 16.513;
   1:L PR[91] R[100]mm/sec CNT100;
   1:  PR[91,1] = PR[90,1] + 11.392;
   1:  PR[91,2] = PR[90,2] + 16.405;
   1:  PR[91,3] = PR[90,3] + 16.519;
   1:L PR[91] R[100]mm/sec CNT100;
   1:  PR[91,1] = PR[90,1] + 10.544;
   1:  PR[91,2] = PR[90,2] + 16.060;
   1:  PR[91,3] = PR[90,3] + 16.525;
   1:L PR[91] R[100]mm/sec CNT100;
   1:  PR[91,1] = PR[90,1] + 9.714;
   1:  PR[91,2] = PR[90,2] + 15.674;
   1:  PR[91,3] = PR[90,3] + 16.532;
   1:L PR[91] R[100]mm/sec CNT100;
   1:  PR[91,1] = PR[90,1] + 8.902;
   1:  PR[91,2] = PR[90,2] + 15.247;
   1:  PR[91,3] = PR[90,3] + 16.538;
   1:L PR[91] R[100]mm/sec CNT100;
   1:  PR[91,1] = PR[90,1] + 8.593;
   1:  PR[91,2] = PR[90,2] + 15.067;
   1:  PR[91,3] = PR[90,3] + 16.544;
   1:L PR[91] R[100]mm/sec CNT100;
   1:  PR[91,1] = PR[90,1] + 8.118;
   1:  PR[91,2] = PR[90,2] + 14.783;
   1:  PR[91,3] = PR[90,3] + 16.546;
   1:L PR[91] R[100]mm/sec CNT100;
   1:  PR[91,1] = PR[90,1] + 7.354;
   1:  PR[91,2] = PR[90,2] + 14.277;
   1:  PR[91,3] = PR[90,3] + 16.550;
   1:L PR[91] R[100]mm/sec CNT100;
   1:  PR[91,1] = PR[90,1] + 6.612;
   1:  PR[91,2] = PR[90,2] + 13.731;
   1:  PR[91,3] = PR[90,3] + 16.556;
   1:L PR[91] R[100]mm/sec CNT100;
   1:  PR[91,1] = PR[90,1] + 5.886;
   1:  PR[91,2] = PR[90,2] + 13.137;
   1:  PR[91,3] = PR[90,3] + 16.563;
   1:L PR[91] R[100]mm/sec CNT100;
   1:  PR[91,1] = PR[90,1] + 5.413;
   1:  PR[91,2] = PR[90,2] + 12.711;
   1:  PR[91,3] = PR[90,3] + 16.569;
   1:L PR[91] R[100]mm/sec CNT100;
   1:  PR[91,1] = PR[90,1] + 4.839;
   1:  PR[91,2] = PR[90,2] + 12.152;
   1:  PR[91,3] = PR[90,3] + 16.573;
   1:L PR[91] R[100]mm/sec CNT100;
   1:  PR[91,1] = PR[90,1] + 4.292;
   1:  PR[91,2] = PR[90,2] + 11.566;
   1:  PR[91,3] = PR[90,3] + 16.579;
   1:L PR[91] R[100]mm/sec CNT100;
   1:  PR[91,1] = PR[90,1] + 3.947;
   1:  PR[91,2] = PR[90,2] + 11.170;
   1:  PR[91,3] = PR[90,3] + 16.584;
   1:L PR[91] R[100]mm/sec CNT100;
   1:  PR[91,1] = PR[90,1] + 3.378;
   1:  PR[91,2] = PR[90,2] + 10.455;
   1:  PR[91,3] = PR[90,3] + 16.588;
   1:L PR[91] R[100]mm/sec CNT100;
   1:  PR[91,1] = PR[90,1] + 2.852;
   1:  PR[91,2] = PR[90,2] + 9.717;
   1:  PR[91,3] = PR[90,3] + 16.594;
   1:L PR[91] R[100]mm/sec CNT100;
   1:  PR[91,1] = PR[90,1] + 2.252;
   1:  PR[91,2] = PR[90,2] + 8.786;
   1:  PR[91,3] = PR[90,3] + 16.600;
   1:L PR[91] R[100]mm/sec CNT100;
   1:  PR[91,1] = PR[90,1] + 1.895;
   1:  PR[91,2] = PR[90,2] + 8.359;
   1:  PR[91,3] = PR[90,3] + 16.607;
   1:L PR[91] R[100]mm/sec CNT100;
   1:  PR[91,1] = PR[90,1] + 1.583;
   1:  PR[91,2] = PR[90,2] + 8.085;
   1:  PR[91,3] = PR[90,3] + 16.611;
   1:L PR[91] R[100]mm/sec CNT100;
   1:  PR[91,1] = PR[90,1] + 1.268;
   1:  PR[91,2] = PR[90,2] + 7.871;
   1:  PR[91,3] = PR[90,3] + 16.614;
   1:L PR[91] R[100]mm/sec CNT100;
   1:  PR[91,1] = PR[90,1] + 0.885;
   1:  PR[91,2] = PR[90,2] + 7.681;
   1:  PR[91,3] = PR[90,3] + 16.617;
   1:L PR[91] R[100]mm/sec CNT100;
   1:  PR[91,1] = PR[90,1] + 0.493;
   1:  PR[91,2] = PR[90,2] + 7.556;
   1:  PR[91,3] = PR[90,3] + 16.619;
   1:L PR[91] R[100]mm/sec CNT100;
   1:  PR[91,1] = PR[90,1] + 0.086;
   1:  PR[91,2] = PR[90,2] + 7.492;
   1:  PR[91,3] = PR[90,3] + 16.622;
   1:L PR[91] R[100]mm/sec CNT100;
   1:  PR[91,1] = PR[90,1] + -0.326;
   1:  PR[91,3] = PR[90,3] + 16.625;
   1:L PR[91] R[100]mm/sec CNT100;
   1:  PR[91,1] = PR[90,1] + -0.733;
   1:  PR[91,2] = PR[90,2] + 7.557;
   1:  PR[91,3] = PR[90,3] + 16.628;
   1:L PR[91] R[100]mm/sec CNT100;
   1:  PR[91,1] = PR[90,1] + -1.126;
   1:  PR[91,2] = PR[90,2] + 7.684;
   1:  PR[91,3] = PR[90,3] + 16.631;
   1:L PR[91] R[100]mm/sec CNT100;
   1:  PR[91,1] = PR[90,1] + -1.507;
   1:  PR[91,2] = PR[90,2] + 7.874;
   1:  PR[91,3] = PR[90,3] + 16.633;
   1:L PR[91] R[100]mm/sec CNT100;
   1:  PR[91,1] = PR[90,1] + -1.822;
   1:  PR[91,2] = PR[90,2] + 8.088;
   1:  PR[91,3] = PR[90,3] + 16.636;
   1:L PR[91] R[100]mm/sec CNT100;
   1:  PR[91,1] = PR[90,1] + -2.133;
   1:  PR[91,2] = PR[90,2] + 8.364;
   1:  PR[91,3] = PR[90,3] + 16.639;
   1:L PR[91] R[100]mm/sec CNT100;
   1:  PR[91,1] = PR[90,1] + -2.494;
   1:  PR[91,2] = PR[90,2] + 8.798;
   1:  PR[91,3] = PR[90,3] + 16.642;
   1:L PR[91] R[100]mm/sec CNT100;
   1:  PR[91,1] = PR[90,1] + -3.089;
   1:  PR[91,2] = PR[90,2] + 9.724;
   1:  PR[91,3] = PR[90,3] + 16.645;
   1:L PR[91] R[100]mm/sec CNT100;
   1:  PR[91,1] = PR[90,1] + -3.522;
   1:  PR[91,2] = PR[90,2] + 10.336;
   1:  PR[91,3] = PR[90,3] + 16.653;
   1:L PR[91] R[100]mm/sec CNT100;
   1:  PR[91,1] = PR[90,1] + -4.182;
   1:  PR[91,2] = PR[90,2] + 11.173;
   1:  PR[91,3] = PR[90,3] + 16.658;
   1:L PR[91] R[100]mm/sec CNT100;
   1:  PR[91,1] = PR[90,1] + -4.791;
   1:  PR[91,2] = PR[90,2] + 11.858;
   1:  PR[91,3] = PR[90,3] + 16.665;
   1:L PR[91] R[100]mm/sec CNT100;
   1:  PR[91,1] = PR[90,1] + -5.075;
   1:  PR[91,2] = PR[90,2] + 12.151;
   1:  PR[91,3] = PR[90,3] + 16.671;
   1:L PR[91] R[100]mm/sec CNT100;
   1:  PR[91,1] = PR[90,1] + -5.435;
   1:  PR[91,2] = PR[90,2] + 12.509;
   1:  PR[91,3] = PR[90,3] + 16.674;
   1:L PR[91] R[100]mm/sec CNT100;
   1:  PR[91,1] = PR[90,1] + -6.124;
   1:  PR[91,2] = PR[90,2] + 13.135;
   1:  PR[91,3] = PR[90,3] + 16.678;
   1:L PR[91] R[100]mm/sec CNT100;
   1:  PR[91,1] = PR[90,1] + -6.874;
   1:  PR[91,2] = PR[90,2] + 13.746;
   1:  PR[91,3] = PR[90,3] + 16.684;
   1:L PR[91] R[100]mm/sec CNT100;
   1:  PR[91,1] = PR[90,1] + -7.592;
   1:  PR[91,2] = PR[90,2] + 14.274;
   1:  PR[91,3] = PR[90,3] + 16.690;
   1:L PR[91] R[100]mm/sec CNT100;
   1:  PR[91,1] = PR[90,1] + -8.159;
   1:  PR[91,2] = PR[90,2] + 14.652;
   1:  PR[91,3] = PR[90,3] + 16.696;
   1:L PR[91] R[100]mm/sec CNT100;
   1:  PR[91,1] = PR[90,1] + -9.144;
   1:  PR[91,2] = PR[90,2] + 15.246;
   1:  PR[91,3] = PR[90,3] + 16.701;
   1:L PR[91] R[100]mm/sec CNT100;
   1:  PR[91,1] = PR[90,1] + -10.223;
   1:  PR[91,2] = PR[90,2] + 15.802;
   1:  PR[91,3] = PR[90,3] + 16.709;
   1:L PR[91] R[100]mm/sec CNT100;
   1:  PR[91,1] = PR[90,1] + -10.785;
   1:  PR[91,2] = PR[90,2] + 16.061;
   1:  PR[91,3] = PR[90,3] + 16.717;
   1:L PR[91] R[100]mm/sec CNT100;
   1:  PR[91,1] = PR[90,1] + -11.634;
   1:  PR[91,2] = PR[90,2] + 16.408;
   1:  PR[91,3] = PR[90,3] + 16.721;
   1:L PR[91] R[100]mm/sec CNT100;
   1:  PR[91,1] = PR[90,1] + -12.492;
   1:  PR[91,2] = PR[90,2] + 16.711;
   1:  PR[91,3] = PR[90,3] + 16.727;
   1:L PR[91] R[100]mm/sec CNT100;
   1:  PR[91,1] = PR[90,1] + -13.361;
   1:  PR[91,2] = PR[90,2] + 16.971;
   1:  PR[91,3] = PR[90,3] + 16.733;
   1:L PR[91] R[100]mm/sec CNT100;
   1:  PR[91,1] = PR[90,1] + -14.239;
   1:  PR[91,2] = PR[90,2] + 17.187;
   1:  PR[91,3] = PR[90,3] + 16.740;
   1:L PR[91] R[100]mm/sec CNT100;
   1:  PR[91,1] = PR[90,1] + -15.128;
   1:  PR[91,2] = PR[90,2] + 17.361;
   1:  PR[91,3] = PR[90,3] + 16.746;
   1:L PR[91] R[100]mm/sec CNT100;
   1:  PR[91,1] = PR[90,1] + -15.426;
   1:  PR[91,2] = PR[90,2] + 17.406;
   1:  PR[91,3] = PR[90,3] + 16.752;
   1:L PR[91] R[100]mm/sec CNT100;
   1:  PR[91,1] = PR[90,1] + -16.017;
   1:  PR[91,2] = PR[90,2] + 17.491;
   1:  PR[91,3] = PR[90,3] + 16.754;
   1:L PR[91] R[100]mm/sec CNT100;
   1:  PR[91,1] = PR[90,1] + -16.913;
   1:  PR[91,2] = PR[90,2] + 17.578;
   1:  PR[91,3] = PR[90,3] + 16.758;
   1:L PR[91] R[100]mm/sec CNT100;
   1:  PR[91,1] = PR[90,1] + -17.779;
   1:  PR[91,2] = PR[90,2] + 17.622;
   1:  PR[91,3] = PR[90,3] + 16.764;
   1:L PR[91] R[100]mm/sec CNT100;
   1:  PR[91,1] = PR[90,1] + -18.599;
   1:  PR[91,2] = PR[90,2] + 17.626;
   1:  PR[91,3] = PR[90,3] + 16.770;
   1:L PR[91] R[100]mm/sec CNT100;
   1:  PR[91,1] = PR[90,1] + -19.732;
   1:  PR[91,2] = PR[90,2] + 17.571;
   1:  PR[91,3] = PR[90,3] + 16.775;
   1:L PR[91] R[100]mm/sec CNT100;
   1:  PR[91,1] = PR[90,1] + -20.252;
   1:  PR[91,2] = PR[90,2] + 17.524;
   1:  PR[91,3] = PR[90,3] + 16.783;
   1:L PR[91] R[100]mm/sec CNT100;
   1:  PR[91,1] = PR[90,1] + -21.080;
   1:  PR[91,2] = PR[90,2] + 17.416;
   1:  PR[91,3] = PR[90,3] + 16.787;
   1:L PR[91] R[100]mm/sec CNT100;
   1:  PR[91,1] = PR[90,1] + -21.903;
   1:  PR[91,2] = PR[90,2] + 17.272;
   1:  PR[91,3] = PR[90,3] + 16.792;
   1:L PR[91] R[100]mm/sec CNT100;
   1:  PR[91,1] = PR[90,1] + -22.535;
   1:  PR[91,2] = PR[90,2] + 17.133;
   1:  PR[91,3] = PR[90,3] + 16.798;
   1:L PR[91] R[100]mm/sec CNT100;
   1:  PR[91,1] = PR[90,1] + -23.454;
   1:  PR[91,2] = PR[90,2] + 16.892;
   1:  PR[91,3] = PR[90,3] + 16.802;
   1:L PR[91] R[100]mm/sec CNT100;
   1:  PR[91,1] = PR[90,1] + -24.341;
   1:  PR[91,2] = PR[90,2] + 16.608;
   1:  PR[91,3] = PR[90,3] + 16.809;
   1:L PR[91] R[100]mm/sec CNT100;
   1:  PR[91,1] = PR[90,1] + -25.164;
   1:  PR[91,2] = PR[90,2] + 16.298;
   1:  PR[91,3] = PR[90,3] + 16.815;
   1:L PR[91] R[100]mm/sec CNT100;
   1:  PR[91,1] = PR[90,1] + -25.969;
   1:  PR[91,2] = PR[90,2] + 15.949;
   1:  PR[91,3] = PR[90,3] + 16.821;
   1:L PR[91] R[100]mm/sec CNT100;
   1:  PR[91,1] = PR[90,1] + -26.754;
   1:  PR[91,2] = PR[90,2] + 15.563;
   1:  PR[91,3] = PR[90,3] + 16.827;
   1:L PR[91] R[100]mm/sec CNT100;
   1:  PR[91,1] = PR[90,1] + -27.215;
   1:  PR[91,2] = PR[90,2] + 15.308;
   1:  PR[91,3] = PR[90,3] + 16.833;
   1:L PR[91] R[100]mm/sec CNT100;
   1:  PR[91,1] = PR[90,1] + -27.515;
   1:  PR[91,2] = PR[90,2] + 15.141;
   1:  PR[91,3] = PR[90,3] + 16.836;
   1:L PR[91] R[100]mm/sec CNT100;
   1:  PR[91,1] = PR[90,1] + -28.255;
   1:  PR[91,2] = PR[90,2] + 14.683;
   1:  PR[91,3] = PR[90,3] + 16.839;
   1:L PR[91] R[100]mm/sec CNT100;
   1:  PR[91,1] = PR[90,1] + -28.968;
   1:  PR[91,2] = PR[90,2] + 14.192;
   1:  PR[91,3] = PR[90,3] + 16.844;
   1:L PR[91] R[100]mm/sec CNT100;
   1:  PR[91,1] = PR[90,1] + -29.654;
   1:  PR[91,2] = PR[90,2] + 13.668;
   1:  PR[91,3] = PR[90,3] + 16.850;
   1:L PR[91] R[100]mm/sec CNT100;
   1:  PR[91,1] = PR[90,1] + -30.311;
   1:  PR[91,2] = PR[90,2] + 13.113;
   1:  PR[91,3] = PR[90,3] + 16.856;
   1:L PR[91] R[100]mm/sec CNT100;
   1:  PR[91,1] = PR[90,1] + -30.938;
   1:  PR[91,2] = PR[90,2] + 12.529;
   1:  PR[91,3] = PR[90,3] + 16.862;
   1:L PR[91] R[100]mm/sec CNT100;
   1:  PR[91,1] = PR[90,1] + -31.534;
   1:  PR[91,2] = PR[90,2] + 11.915;
   1:  PR[91,3] = PR[90,3] + 16.868;
   1:L PR[91] R[100]mm/sec CNT100;
   1:  PR[91,1] = PR[90,1] + -32.108;
   1:  PR[91,2] = PR[90,2] + 11.261;
   1:  PR[91,3] = PR[90,3] + 16.874;
   1:L PR[91] R[100]mm/sec CNT100;
   1:  PR[91,1] = PR[90,1] + -32.626;
   1:  PR[91,2] = PR[90,2] + 10.607;
   1:  PR[91,3] = PR[90,3] + 16.879;
   1:L PR[91] R[100]mm/sec CNT100;
   1:  PR[91,1] = PR[90,1] + -33.119;
   1:  PR[91,2] = PR[90,2] + 9.914;
   1:  PR[91,3] = PR[90,3] + 16.885;
   1:L PR[91] R[100]mm/sec CNT100;
   1:  PR[91,1] = PR[90,1] + -33.577;
   1:  PR[91,2] = PR[90,2] + 9.198;
   1:  PR[91,3] = PR[90,3] + 16.891;
   1:L PR[91] R[100]mm/sec CNT100;
   1:  PR[91,1] = PR[90,1] + -33.999;
   1:  PR[91,2] = PR[90,2] + 8.462;
   1:  PR[91,3] = PR[90,3] + 16.897;
   1:L PR[91] R[100]mm/sec CNT100;
   1:  PR[91,1] = PR[90,1] + -34.383;
   1:  PR[91,2] = PR[90,2] + 7.708;
   1:  PR[91,3] = PR[90,3] + 16.902;
   1:L PR[91] R[100]mm/sec CNT100;
   1:  PR[91,1] = PR[90,1] + -34.729;
   1:  PR[91,2] = PR[90,2] + 6.941;
   1:  PR[91,3] = PR[90,3] + 16.908;
   1:L PR[91] R[100]mm/sec CNT100;
   1:  PR[91,1] = PR[90,1] + -35.036;
   1:  PR[91,2] = PR[90,2] + 6.164;
   1:  PR[91,3] = PR[90,3] + 16.914;
   1:L PR[91] R[100]mm/sec CNT100;
   1:  PR[91,1] = PR[90,1] + -35.304;
   1:  PR[91,2] = PR[90,2] + 5.379;
   1:  PR[91,3] = PR[90,3] + 16.919;
   1:L PR[91] R[100]mm/sec CNT100;
   1:  PR[91,1] = PR[90,1] + -35.530;
   1:  PR[91,2] = PR[90,2] + 4.586;
   1:  PR[91,3] = PR[90,3] + 16.925;
   1:L PR[91] R[100]mm/sec CNT100;
   1:  PR[91,1] = PR[90,1] + -35.716;
   1:  PR[91,2] = PR[90,2] + 3.784;
   1:  PR[91,3] = PR[90,3] + 16.931;
   1:L PR[91] R[100]mm/sec CNT100;
   1:  PR[91,1] = PR[90,1] + -35.861;
   1:  PR[91,2] = PR[90,2] + 2.971;
   1:  PR[91,3] = PR[90,3] + 16.936;
   1:L PR[91] R[100]mm/sec CNT100;
   1:  PR[91,1] = PR[90,1] + -35.965;
   1:  PR[91,2] = PR[90,2] + 2.143;
   1:  PR[91,3] = PR[90,3] + 16.942;
   1:L PR[91] R[100]mm/sec CNT100;
   1:  PR[91,1] = PR[90,1] + -36.028;
   1:  PR[91,2] = PR[90,2] + 1.295;
   1:  PR[91,3] = PR[90,3] + 16.947;
   1:L PR[91] R[100]mm/sec CNT100;
   1:  PR[91,1] = PR[90,1] + -36.051;
   1:  PR[91,2] = PR[90,2] + 0.428;
   1:  PR[91,3] = PR[90,3] + 16.953;
   1:L PR[91] R[100]mm/sec CNT100;
   1:  PR[91,1] = PR[90,1] + -36.028;
   1:  PR[91,2] = PR[90,2] + -0.440;
   1:  PR[91,3] = PR[90,3] + 16.959;
   1:L PR[91] R[100]mm/sec CNT100;
   1:  PR[91,1] = PR[90,1] + -35.965;
   1:  PR[91,2] = PR[90,2] + -1.288;
   1:  PR[91,3] = PR[90,3] + 16.965;
   1:L PR[91] R[100]mm/sec CNT100;
   1:  PR[91,1] = PR[90,1] + -35.861;
   1:  PR[91,2] = PR[90,2] + -2.116;
   1:  PR[91,3] = PR[90,3] + 16.971;
   1:L PR[91] R[100]mm/sec CNT100;
   1:  PR[91,1] = PR[90,1] + -35.716;
   1:  PR[91,2] = PR[90,2] + -2.929;
   1:  PR[91,3] = PR[90,3] + 16.976;
   1:L PR[91] R[100]mm/sec CNT100;
   1:  PR[91,1] = PR[90,1] + -35.530;
   1:  PR[91,2] = PR[90,2] + -3.731;
   1:  PR[91,3] = PR[90,3] + 16.982;
   1:L PR[91] R[100]mm/sec CNT100;
   1:  PR[91,1] = PR[90,1] + -35.304;
   1:  PR[91,2] = PR[90,2] + -4.524;
   1:  PR[91,3] = PR[90,3] + 16.987;
   1:L PR[91] R[100]mm/sec CNT100;
   1:  PR[91,1] = PR[90,1] + -35.036;
   1:  PR[91,2] = PR[90,2] + -5.309;
   1:  PR[91,3] = PR[90,3] + 16.993;
   1:L PR[91] R[100]mm/sec CNT100;
   1:  PR[91,1] = PR[90,1] + -34.729;
   1:  PR[91,2] = PR[90,2] + -6.086;
   1:  PR[91,3] = PR[90,3] + 16.998;
   1:L PR[91] R[100]mm/sec CNT100;
   1:  PR[91,1] = PR[90,1] + -34.383;
   1:  PR[91,2] = PR[90,2] + -6.853;
   1:  PR[91,3] = PR[90,3] + 17.004;
   1:L PR[91] R[100]mm/sec CNT100;
   1:  PR[91,1] = PR[90,1] + -33.999;
   1:  PR[91,2] = PR[90,2] + -7.607;
   1:  PR[91,3] = PR[90,3] + 17.010;
   1:L PR[91] R[100]mm/sec CNT100;
   1:  PR[91,1] = PR[90,1] + -33.577;
   1:  PR[91,2] = PR[90,2] + -8.343;
   1:  PR[91,3] = PR[90,3] + 17.016;
   1:L PR[91] R[100]mm/sec CNT100;
   1:  PR[91,1] = PR[90,1] + -33.119;
   1:  PR[91,2] = PR[90,2] + -9.059;
   1:  PR[91,3] = PR[90,3] + 17.021;
   1:L PR[91] R[100]mm/sec CNT100;
   1:  PR[91,1] = PR[90,1] + -32.626;
   1:  PR[91,2] = PR[90,2] + -9.751;
   1:  PR[91,3] = PR[90,3] + 17.027;
   1:L PR[91] R[100]mm/sec CNT100;
   1:  PR[91,1] = PR[90,1] + -32.098;
   1:  PR[91,2] = PR[90,2] + -10.419;
   1:  PR[91,3] = PR[90,3] + 17.033;
   1:L PR[91] R[100]mm/sec CNT100;
   1:  PR[91,1] = PR[90,1] + -31.534;
   1:  PR[91,2] = PR[90,2] + -11.060;
   1:  PR[91,3] = PR[90,3] + 17.038;
   1:L PR[91] R[100]mm/sec CNT100;
   1:  PR[91,1] = PR[90,1] + -30.938;
   1:  PR[91,2] = PR[90,2] + -11.674;
   1:  PR[91,3] = PR[90,3] + 17.044;
   1:L PR[91] R[100]mm/sec CNT100;
   1:  PR[91,1] = PR[90,1] + -30.311;
   1:  PR[91,2] = PR[90,2] + -12.258;
   1:  PR[91,3] = PR[90,3] + 17.050;
   1:L PR[91] R[100]mm/sec CNT100;
   1:  PR[91,1] = PR[90,1] + -29.654;
   1:  PR[91,2] = PR[90,2] + -12.813;
   1:  PR[91,3] = PR[90,3] + 17.056;
   1:L PR[91] R[100]mm/sec CNT100;
   1:  PR[91,1] = PR[90,1] + -28.968;
   1:  PR[91,2] = PR[90,2] + -13.337;
   1:  PR[91,3] = PR[90,3] + 17.062;
   1:L PR[91] R[100]mm/sec CNT100;
   1:  PR[91,1] = PR[90,1] + -28.254;
   1:  PR[91,2] = PR[90,2] + -13.828;
   1:  PR[91,3] = PR[90,3] + 17.067;
   1:L PR[91] R[100]mm/sec CNT100;
   1:  PR[91,1] = PR[90,1] + -27.897;
   1:  PR[91,2] = PR[90,2] + -14.051;
   1:  PR[91,3] = PR[90,3] + 17.073;
   1:L PR[91] R[100]mm/sec CNT100;
   1:  PR[91,1] = PR[90,1] + -27.517;
   1:  PR[91,2] = PR[90,2] + -14.285;
   1:  PR[91,3] = PR[90,3] + 17.076;
   1:L PR[91] R[100]mm/sec CNT100;
   1:  PR[91,1] = PR[90,1] + -26.754;
   1:  PR[91,2] = PR[90,2] + -14.708;
   1:  PR[91,3] = PR[90,3] + 17.079;
   1:L PR[91] R[100]mm/sec CNT100;
   1:  PR[91,1] = PR[90,1] + -25.969;
   1:  PR[91,2] = PR[90,2] + -15.094;
   1:  PR[91,3] = PR[90,3] + 17.085;
   1:L PR[91] R[100]mm/sec CNT100;
   1:  PR[91,1] = PR[90,1] + -25.164;
   1:  PR[91,2] = PR[90,2] + -15.443;
   1:  PR[91,3] = PR[90,3] + 17.091;
   1:L PR[91] R[100]mm/sec CNT100;
   1:  PR[91,1] = PR[90,1] + -24.320;
   1:  PR[91,2] = PR[90,2] + -15.760;
   1:  PR[91,3] = PR[90,3] + 17.097;
   1:L PR[91] R[100]mm/sec CNT100;
   1:  PR[91,1] = PR[90,1] + -23.532;
   1:  PR[91,2] = PR[90,2] + -16.014;
   1:  PR[91,3] = PR[90,3] + 17.103;
   1:L PR[91] R[100]mm/sec CNT100;
   1:  PR[91,1] = PR[90,1] + -22.537;
   1:  PR[91,2] = PR[90,2] + -16.277;
   1:  PR[91,3] = PR[90,3] + 17.109;
   1:L PR[91] R[100]mm/sec CNT100;
   1:  PR[91,1] = PR[90,1] + -21.605;
   1:  PR[91,2] = PR[90,2] + -16.472;
